Yaskawa INFORM job: SKRZYNIA_5240_180_STOPNI_10B_NEW.JBI

/JOB
//NAME SKRZYNIA_5240_180_STOPNI_10B_NEW
///FOLDERNAME 02-SKRZYNIE_JOBS
//POS
///NPOS 773,773,0,34,0,0
///TOOL 0
///POSTYPE PULSE
///PULSE
C00000=-21231,-51303,42314,2367,6591,-1439
C00001=-12854,-61498,-6635,149088,-29435,16513
C00002=84284,-61498,-6635,149088,14842,16513
C00003=84426,-61498,-62039,149088,14842,16513
C00004=84426,-61498,-83719,149088,14842,16513
C00005=40079,-25830,-61904,72398,37828,17494
C00006=40079,-25830,-61904,72398,37828,17494
C00007=38824,-23395,-60038,72349,38727,17731
C00008=41545,-22667,-59464,70826,37145,18191
C00009=40079,-25830,-61904,72398,37828,17494
C00010=40079,-23879,-31232,97616,36989,2612
C00011=40241,-22903,-30855,97033,36795,2952
C00012=39596,-21803,-29985,96678,37187,3182
C00013=41542,-21522,-29763,96797,35874,3054
C00014=40241,-22903,-30855,97033,36795,2952
C00015=44500,-22967,-34027,49689,40772,15208
C00016=44759,-21950,-33222,49364,40770,15399
C00017=43898,-20603,-32137,49608,41392,15289
C00018=45676,-20288,-31878,48567,40497,15854
C00019=44759,-21950,-33222,49364,40770,15399
C00020=50639,-31838,-53853,40430,42590,20636
C00021=47737,-42531,-47731,84740,46626,-3202
C00022=73324,-51450,-15857,136644,48513,-27329
C00023=28578,-31257,-33285,101874,54895,-3139
C00024=29101,-23166,-41439,93785,52323,3372
C00025=30342,-16402,-40775,90158,51109,6027
C00026=29555,-14242,-38855,90054,51607,6222
C00027=31304,-14182,-38798,89754,50458,6198
C00028=30342,-16402,-40775,90158,51109,6027
C00029=37840,-26567,-47806,97824,39338,5403
C00030=38314,-22656,-45541,96192,38787,6352
C00031=38740,-21749,-44817,95954,38481,6451
C00032=38106,-20505,-43805,95701,38856,6673
C00033=39920,-20274,-43616,95549,37666,6573
C00034=38740,-21749,-44817,95954,38481,6451
C00035=35154,-23288,-28184,89821,43405,2441
C00036=35403,-21021,-26397,89340,43215,2751
C00037=34678,-19569,-25213,89063,43699,2948
C00038=36545,-19419,-25091,89018,42427,2940
C00039=35403,-21021,-26397,89340,43215,2751
C00040=46673,-28267,-59493,36306,49500,22578
C00041=47298,-25083,-54483,36432,48421,22382
C00042=46134,-23276,-53085,36983,49197,22170
C00043=48093,-22778,-52692,35651,48513,22818
C00044=47298,-25083,-54483,36432,48421,22382
C00045=43000,-32780,-49011,53703,41088,15214
C00046=66148,-65994,-55487,105361,28212,-7739
C00047=66148,-65994,-55487,105361,28212,-7739
C00048=59848,-54778,-49507,133915,29212,-10807
C00049=45497,-38347,-41839,114412,32622,-465
C00050=46376,-32635,-46933,102993,29107,5780
C00051=46303,-28031,-46898,97061,28371,8976
C00052=45038,-26161,-45521,96183,29128,9541
C00053=46946,-25787,-45238,96120,27855,9431
C00054=46303,-28031,-46898,97061,28371,8976
C00055=45864,-17128,1685,129467,40696,-9274
C00056=46023,-15894,1830,128891,40053,-8896
C00057=45181,-14790,2774,128176,40341,-8535
C00058=46921,-14545,2986,129317,39465,-9073
C00059=45402,-17127,796,128656,40504,-8810
C00060=42828,-21985,-11573,106778,34538,-1929
C00061=43349,-21404,-11124,106831,34165,-1930
C00062=42250,-19876,-9917,105946,34757,-1485
C00063=44494,-19460,-9583,106781,33302,-1837
C00064=42797,-21858,-11474,106726,34550,-1903
C00065=42956,-14057,7354,88292,32197,-569
C00066=43438,-13569,7781,88275,31880,-510
C00067=42549,-12302,8904,87823,32462,-349
C00068=44721,-11883,9282,88161,31033,-316
C00069=42944,-14884,6642,88491,32210,-682
C00070=42956,-14057,7354,88292,32197,-569
C00071=43438,-13569,7781,88275,31880,-510
C00072=42549,-12302,8904,87823,32462,-349
C00073=44721,-11883,9282,88161,31033,-316
C00074=42944,-14884,6642,88491,32210,-682
C00075=42492,-36415,-29790,92406,42740,11684
C00076=29699,-14901,-14062,86637,51249,15251
C00077=28921,-12904,-12269,86425,51786,15406
C00078=30978,-12767,-12144,86426,50380,15429
C00079=29506,-17416,-16239,86937,51377,15018
C00080=29523,-100,37175,104016,54946,1530
C00081=29670,3692,41450,104134,54886,1470
C00082=29289,4768,42714,104010,55127,1477
C00083=31025,4720,42655,104739,54116,1295
C00084=29634,3577,41316,104108,54910,1473
C00085=88410,-69609,-60867,139529,19008,-8209
C00086=82254,-59190,-37505,135829,26015,-2584
C00087=48709,-26647,-10027,118963,31871,904
C00088=44740,-24992,-19428,105622,30913,8023
C00089=35836,-10089,175,120717,54219,3716
C00090=33571,-11609,-5533,116057,52820,8482
C00091=32638,-9483,-3533,115639,53262,8773
C00092=34483,-9329,-3384,116184,52162,8425
C00093=33571,-11609,-5533,116057,52820,8482
C00094=29299,-14235,-8112,85858,51306,13749
C00095=30258,-13056,-7056,85778,50658,13854
C00096=29454,-11053,-5212,85557,51212,13988
C00097=31306,-10982,-5149,85624,49953,14016
C00098=30258,-13056,-7056,85778,50658,13854
C00099=44150,-27478,-14760,79983,38437,11062
C00100=60260,-41997,-20174,82745,25327,6782
C00101=62412,-62489,-12046,-12266,17816,34850
C00102=0,-52280,40443,0,6876,0
C00103=-681,-52632,38645,-5695,5489,-631
C00104=-17840,-61498,-6635,-149088,-29435,-16513
C00105=-84284,-61498,-6635,-149088,14842,-16513
C00106=-84426,-61498,-62039,-149088,14842,-16513
C00107=-84426,-61498,-83719,-149088,14842,-16513
C00108=-83351,-27062,-60322,-167360,37385,6517
C00109=-83351,-27062,-60322,-167360,37385,23281
C00110=-45097,-23850,-79932,-76262,26943,-22849
C00111=-48253,-15729,-73342,-71138,25693,-24842
C00112=-50302,-13076,-73239,-65836,25323,-27140
C00113=-49401,-11675,-71961,-66260,25816,-27133
C00114=-50608,-11574,-71867,-65226,25249,-27391
C00115=-49660,-13361,-73494,-66442,25615,-26975
C00116=-48242,-21102,-77802,-73044,25430,-23851
C00117=-42432,-29691,-46140,-101591,34194,-3953
C00118=-40467,-32259,-45349,-89481,35752,-6083
C00119=-35590,-22323,-38089,-87474,43148,-7978
C00120=-34853,-20780,-36847,-87247,43643,-8181
C00121=-37029,-20471,-36594,-86926,42180,-8224
C00122=-35503,-23333,-38886,-87700,43207,-7835
C00123=-41659,-25848,-37197,-61468,39541,-12344
C00124=-42019,-23363,-32043,-63110,38591,-11327
C00125=-41283,-22167,-31102,-63128,39154,-11341
C00126=-43189,-21868,-30866,-62281,38009,-11788
C00127=-40846,-25460,-35158,-62968,39555,-11455
C00128=-39561,-32409,-42051,-71473,38885,-9254
C00129=-88477,-67032,-53890,-125185,13082,17955
C00130=-90715,-66667,-50935,-152816,24533,28486
C00131=-30735,-26920,-32844,-95116,50209,-1071
C00132=-37180,-24683,-31930,-114741,47007,2943
C00133=-36407,-19634,-34656,-109847,45004,-453
C00134=-38352,-16604,-33863,-108521,43129,-1176
C00135=-37479,-14809,-32279,-108169,43576,-1482
C00136=-39395,-14487,-31992,-108361,42368,-1194
C00137=-37253,-18321,-35339,-108644,43916,-1187
C00138=-30948,-19486,-27368,-89515,49970,-2899
C00139=-32453,-17458,-25663,-89179,48933,-3088
C00140=-31896,-16151,-24534,-89028,49305,-3221
C00141=-33527,-16125,-24510,-88960,48196,-3202
C00142=-31291,-18911,-26892,-89421,49733,-2955
C00143=-32789,-14788,-10714,-75998,48642,-1904
C00144=-33953,-13481,-9550,-75758,47902,-2112
C00145=-33380,-12226,-8408,-75670,48319,-2157
C00146=-35020,-12164,-8351,-75529,47228,-2306
C00147=-33300,-14767,-10697,-75957,48300,-1949
C00148=-33300,-14767,-10697,-75957,48300,-1949
C00149=-33901,-13199,-7224,-76945,47663,-1266
C00150=-33178,-11617,-5779,-76815,48184,-1329
C00151=-35129,-11426,-5603,-76688,46886,-1497
C00152=-32900,-14718,-9841,-76444,48459,-1584
C00153=-46324,-38325,-53351,-48650,39022,-16558
C00154=-84678,-53272,-42524,-56273,5220,-14251
C00155=-79949,-57830,-54545,-43165,18800,-25262
C00156=-85199,-63426,-59279,-35356,8253,-25340
C00157=-43240,-40066,-69296,-76804,34492,-13950
C00158=-32352,-24302,-62495,-76398,48702,-17646
C00159=-33867,-19497,-59989,-74208,48202,-18898
C00160=-33043,-17469,-58279,-74274,48770,-19034
C00161=-35172,-17180,-58031,-73305,47532,-19251
C00162=-33150,-20833,-61090,-74721,48572,-18687
C00163=-32525,-19963,-22291,-97454,48417,-2656
C00164=-34479,-17146,-19937,-97221,47013,-2812
C00165=-33716,-15515,-18525,-96928,47480,-3025
C00166=-35357,-15455,-18472,-97073,46375,-2908
C00167=-33341,-18474,-21063,-97306,47817,-2759
C00168=-32838,-10388,7981,-94473,48357,2926
C00169=-33747,-9461,8037,-94117,47673,2571
C00170=-33094,-8062,9377,-93861,48090,2458
C00171=-34952,-7927,9507,-94260,46861,2543
C00172=-33010,-10379,7174,-94037,48174,2591
C00173=-36099,-20774,-22249,-70758,44565,-7624
C00174=-37926,-16067,-12890,-73276,42575,-5996
C00175=-37323,-14944,-11908,-73188,43017,-6038
C00176=-39053,-14785,-11769,-72915,41882,-6255
C00177=-37847,-19214,-17221,-72670,42783,-6386
C00178=-36099,-20774,-22249,-70758,44565,-7624
C00179=-37926,-16067,-12890,-73276,42575,-5996
C00180=-37323,-14944,-11908,-73188,43017,-6038
C00181=-39053,-14785,-11769,-72915,41882,-6255
C00182=-37847,-19214,-17221,-72670,42783,-6386
C00183=-36099,-20774,-22249,-70758,44565,-7624
C00184=-37926,-16067,-12890,-73276,42575,-5996
C00185=-37323,-14944,-11908,-73188,43017,-6038
C00186=-39053,-14785,-11769,-72915,41882,-6255
C00187=-37847,-19214,-17221,-72670,42783,-6386
C00188=-37874,14907,75180,-111692,46453,18697
C00189=-37834,19259,81880,-112749,47050,19446
C00190=-37304,21381,85363,-113034,47644,19820
C00191=-39330,21904,86247,-114552,46854,20222
C00192=-38061,19744,82664,-113035,47027,19575
C00193=-73757,-59015,-49060,-81128,17325,-3444
C00194=-59391,-59726,-723,-139936,47315,26256
C00195=-59391,-63256,-7305,-138930,45803,25558
C00196=-41911,-25348,-18707,-96909,37821,5942
C00197=-39278,-18921,-13723,-94727,39374,4724
C00198=-50267,-3803,20766,-145166,53580,20077
C00199=-49199,-2294,22340,-144514,53890,19722
C00200=-50839,-1881,22778,-145489,53339,20243
C00201=-50267,-457,30009,-146420,56926,21139
C00202=-39278,-18921,-13723,-94727,39374,4724
C00203=-38355,-17353,-12416,-94258,39960,4466
C00204=-40180,-17161,-12255,-94505,38724,4557
C00205=-37963,-22229,-16363,-95272,40353,5112
C00206=-56568,-73357,-35482,-123268,35826,13545
C00207=-46099,-67236,-11725,-98004,28606,19827
C00208=275,-40498,62911,330,272,-175
C00209=-21231,-51303,42314,2367,6591,-1439
C00210=-12854,-61498,-6635,149088,-29435,16513
C00211=84284,-61498,-6635,149088,14842,16513
C00212=84426,-61498,-62039,149088,14842,16513
C00213=84426,-61498,-83719,149088,14842,16513
C00214=40079,-25830,-61904,72398,37828,17494
C00215=38665,-12403,-32409,107781,42694,-4781
C00216=38665,-12616,-38699,103566,41336,-2086
C00217=40079,-23879,-31232,97616,36989,2612
C00218=41034,-22333,-61710,53029,45515,35529
C00219=41034,-23109,-56119,56672,43067,33108
C00220=40241,-22903,-30855,97033,36795,2952
C00221=44500,-24561,-52671,41420,48760,20730
C00222=37674,-15115,-44130,49660,57471,17042
C00223=37674,-15093,-37691,51888,54769,15111
C00224=44759,-23105,-42292,45130,44325,18129
C00225=50639,-31838,-53853,40430,42590,20636
C00226=47737,-42531,-47731,84740,46626,-3202
C00227=78713,-49095,-28754,133607,38203,-24422
C00228=28578,-31257,-33285,101874,54895,-3139
C00229=29101,-23166,-41439,93785,52323,3372
C00230=31163,-13587,-30677,93779,50972,3168
C00231=31163,-14026,-37120,90592,50610,5586
C00232=30342,-16304,-38140,91492,51220,5006
C00233=37840,-26567,-47806,97824,39338,5403
C00234=38314,-22656,-45541,96192,38787,6352
C00235=39658,-19732,-37407,100215,38572,3786
C00236=39658,-20175,-43840,95284,37805,6758
C00237=38740,-21749,-44817,95954,38481,6451
C00238=35154,-25126,-38164,84243,43431,6092
C00239=35628,-20373,-48281,63877,49123,23186
C00240=35628,-20245,-42140,67132,47541,20849
C00241=35403,-21021,-26397,89340,43215,2751
C00242=46673,-26636,-70072,32738,56435,25418
C00243=35383,-13840,-53792,49898,63478,22502
C00244=35383,-14670,-48593,51546,60904,20775
C00245=47298,-24788,-58951,34834,51068,23565
C00246=43000,-32780,-49011,53703,41088,15214
C00247=90538,-65158,-52413,145953,6697,-22013
C00248=90538,-65158,-52413,145953,6697,-22013
C00249=59848,-54778,-49507,133915,29212,-10807
C00250=45497,-38347,-41839,114412,32622,-465
C00251=46376,-32635,-46933,102993,29107,5780
C00252=33967,-11360,-33206,103445,48358,510
C00253=33967,-11425,-39323,99951,47288,2995
C00254=46303,-28031,-46898,97061,28371,8976
C00255=45864,-24383,-22135,118487,33937,-2761
C00256=34441,-6148,1727,116719,55152,-8810
C00257=34441,-8494,-7364,114007,52974,-6586
C00258=45402,-26628,-33163,110407,31435,1774
C00259=42828,-30834,-56687,70923,33806,18230
C00260=32432,-16862,-57229,61149,56469,35022
C00261=32432,-17753,-51657,63804,54519,32761
C00262=42797,-29457,-43215,82997,32293,11437
C00263=42956,-27250,-43688,55004,39651,18538
C00264=34828,-16613,-38353,58296,54652,20387
C00265=34828,-16027,-31548,60910,52619,18267
C00266=33058,-19049,-34141,61806,53461,17709
C00267=33058,-12296,-3124,73891,47808,8644
C00268=33058,-12296,-3124,73891,47808,8644
C00269=34828,-9500,-717,73395,46757,9098
C00270=34828,-6540,9127,77476,45790,6283
C00271=33897,-9329,6906,77965,46306,5856
C00272=33897,-9329,6906,77965,46306,5856
C00273=34828,-9385,-322,73557,46711,8985
C00274=34828,-6437,9450,77608,45767,6193
C00275=34037,-8372,7553,77721,46264,6039
C00276=34037,3206,39942,90427,45468,-2620
C00277=34037,-4564,18961,82315,45612,2890
C00278=34657,-86,29234,85939,44999,527
C00279=34657,5122,42910,91205,45125,-3022
C00280=29506,-17416,-16239,86937,51377,15018
C00281=88410,-69609,-60867,139529,19008,-8209
C00282=82254,-59190,-37505,135829,26015,-2584
C00283=48709,-26647,-10027,118963,31871,904
C00284=44740,-24992,-19428,105622,30913,8023
C00285=35836,-628,28594,126575,61828,-1622
C00286=32584,7682,39174,123909,66904,-2731
C00287=32584,2860,25722,121968,63529,-448
C00288=33571,-6628,11088,120434,56899,4821
C00289=29299,-14235,-8112,85858,51306,13749
C00290=31207,-8871,1432,87980,49993,12258
C00291=31207,-5884,11163,91534,50189,9605
C00292=30258,-13056,-7056,85778,50658,13854
C00293=44150,-27478,-14760,79983,38437,11062
C00294=60260,-41997,-20174,82745,25327,6782
C00295=62412,-62489,-12046,-12266,17816,34850
C00296=0,-52280,40443,0,6876,0
C00297=-681,-52632,38645,-5695,5489,-631
C00298=-17840,-61498,-6635,-149088,-29435,-16513
C00299=-84284,-61498,-6635,-149088,14842,-16513
C00300=-84426,-61498,-62039,-149088,14842,-16513
C00301=-84426,-61498,-83719,-149088,14842,-16513
C00302=-83351,-27062,-60322,-167360,37385,6517
C00303=-83351,-27062,-60322,-167360,37385,23281
C00304=-45097,-23850,-79932,-76262,26943,-22849
C00305=-48253,-15729,-73342,-71138,25693,-24842
C00306=-42968,-5377,-68871,-73541,34127,-27123
C00307=-42968,-1764,-72258,-66870,35661,-30967
C00308=-49660,-13361,-73494,-66442,25615,-26975
C00309=-48242,-21102,-77802,-73044,25430,-23851
C00310=-42432,-29691,-46140,-101591,34194,-3953
C00311=-40467,-32259,-45349,-89481,35752,-6083
C00312=-32572,-16306,-55553,-67397,53381,-30018
C00313=-32572,-17083,-50158,-70353,51979,-27676
C00314=-35503,-23333,-38886,-87700,43207,-7835
C00315=-41659,-27404,-51576,-53376,44034,-17488
C00316=-31493,-12293,-40596,-60462,61580,-18646
C00317=-31493,-12246,-34421,-62460,59687,-16660
C00318=-40846,-26766,-43924,-57962,41907,-14588
C00319=-39561,-32409,-42051,-71473,38885,-9254
C00320=-88477,-67032,-53890,-125185,13082,17955
C00321=-90715,-66667,-50935,-152816,24533,28486
C00322=-30735,-26920,-32844,-95116,50209,-1071
C00323=-37180,-24683,-31930,-114741,47007,2943
C00324=-36407,-19634,-34656,-109847,45004,-453
C00325=-39265,-13210,-22525,-113458,44747,2144
C00326=-39265,-14219,-29616,-109727,42998,-318
C00327=-37253,-17754,-30753,-111100,44998,450
C00328=-30948,-19486,-27368,-89515,49970,-2899
C00329=-32883,-16993,-41795,-70354,52410,-19465
C00330=-32883,-16648,-35340,-73373,51262,-17121
C00331=-31291,-18911,-26892,-89421,49733,-2955
C00332=-32789,-18082,-25081,-70149,50526,-6217
C00333=-30947,-8963,-19167,-66964,58291,-13111
C00334=-30947,-7534,-11276,-69435,56821,-10881
C00335=-33300,-16430,-17409,-73196,49065,-3948
C00336=-33300,-18454,-27193,-69159,50560,-6941
C00337=-29440,-7196,-21034,-66741,61979,-14499
C00338=-29440,-6022,-13253,-68913,60441,-12298
C00339=-32900,-16744,-17947,-73145,49365,-3984
C00340=-46324,-38325,-53351,-48650,39022,-16558
C00341=-84678,-53272,-42524,-56273,5220,-14251
C00342=-79949,-57830,-54545,-43165,18800,-25262
C00343=-85199,-63426,-59279,-35356,8253,-25340
C00344=-43240,-40066,-69296,-76804,34492,-13950
C00345=-32352,-24302,-62495,-76398,48702,-17646
C00346=-32091,-8283,-47690,-89191,50586,-9020
C00347=-32091,-6854,-52880,-85538,50580,-11777
C00348=-33150,-19215,-66726,-70659,49900,-21662
C00349=-32525,-23315,-42550,-87560,47339,-9680
C00350=-33177,-11430,-23623,-100299,50817,3381
C00351=-33177,-12228,-30638,-97022,49957,920
C00352=-33341,-22016,-46198,-84312,46879,-11867
C00353=-32838,-21830,-40242,-73680,49831,-12021
C00354=-32060,-14432,-37779,-68594,55292,-20152
C00355=-32060,-13998,-31234,-71279,54006,-17916
C00356=-32826,-17642,-34445,-71437,53361,-17708
C00357=-36099,-24001,-62103,-52600,56003,-20988
C00358=-33061,-10268,-52363,-54704,65882,-25434
C00359=-33061,-11342,-46906,-56402,63410,-23481
C00360=-32436,-13964,-49327,-56793,63580,-23241
C00361=-36099,-22018,-27900,-68071,45501,-9434
C00362=-33133,-10810,-21932,-64736,55524,-15558
C00363=-33133,-9463,-14247,-67406,53929,-13330
C00364=-32817,-11797,-16457,-67620,54048,-13161
C00365=-36099,-9367,15363,-88420,42122,3838
C00366=-33275,421,22196,-80432,49557,-3328
C00367=-33275,4923,34904,-84824,49106,-106
C00368=-32887,2565,32173,-84656,49359,-162
C00369=-32887,2565,32173,-84656,49359,-162
C00370=-33016,5847,38022,-85966,49224,775
C00371=-33016,12470,54924,-91440,49393,4788
C00372=-31218,6775,44553,-88539,50343,3051
C00373=-82794,-53123,-36553,-147152,20085,23769
C00374=-59391,-59726,-723,-139936,47315,26256
C00375=-59391,-69594,-18878,-137021,43274,24283
C00376=-41911,-25348,-18707,-96909,37821,5942
C00377=-39278,-18921,-13723,-94727,39374,4724
C00378=-42007,14667,57624,-137771,70069,18031
C00379=-42007,7816,40199,-136118,64730,15895
C00380=-50267,-457,30009,-146420,56926,21139
C00381=-32199,-12839,-21112,-74266,52126,-18055
C00382=-32186,-11312,-13395,-77340,51278,-15674
C00383=-37963,-22229,-16363,-95272,40353,5112
C00384=-66368,-73811,-34662,-141094,38161,28545
C00385=-46099,-67236,-11725,-98004,28606,19827
C00386=275,-40498,62911,330,272,-175
C00387=-21231,-51303,42314,2367,6591,-1439
C00388=-12854,-61498,-6635,149088,-29435,16513
C00389=32880,-72586,-50560,79734,53940,25582
C00390=76664,-93599,-96338,114349,24908,7990
C00391=72545,-76403,-90681,98079,12187,16258
C00392=68435,-42241,-79282,43384,21203,43145
C00393=65057,-16377,-54230,51764,24572,24912
C00394=65057,-16377,-54230,51764,24572,24912
C00395=63338,-14509,-52578,53100,25585,24479
C00396=65493,-13068,-51269,50530,24633,25485
C00397=65057,-16377,-54230,51764,24572,24912
C00398=65057,-15356,-24189,99795,20011,765
C00399=64877,-14372,-23690,98704,20045,1316
C00400=64002,-13489,-22890,98156,20604,1621
C00401=65592,-12702,-22173,98357,19527,1466
C00402=64877,-14372,-23690,98704,20045,1316
C00403=68341,-13254,-25781,29903,31229,25524
C00404=68283,-12212,-24821,29865,31356,25548
C00405=67188,-11145,-23825,30867,31841,25051
C00406=68624,-10377,-23095,29361,31405,25809
C00407=68283,-12212,-24821,29865,31356,25548
C00408=67373,-28813,-51747,26561,36937,27500
C00409=65665,-56911,-59086,75825,31170,1181
C00410=86238,-56758,-47218,93606,16664,-7096
C00411=86238,-56758,-47218,93606,16664,-7096
C00412=58162,-25487,-29222,106212,35121,-6052
C00413=54729,-17550,-36821,90686,35172,3055
C00414=53879,-10723,-35593,84994,35691,6442
C00415=52628,-8898,-33837,85063,36512,6546
C00416=54193,-8333,-33282,84633,35489,6620
C00417=53879,-10723,-35593,84994,35691,6442
C00418=63265,-18185,-41125,95483,22448,4389
C00419=62561,-14368,-38517,92984,22773,5727
C00420=62689,-13396,-37636,92694,22678,5861
C00421=61812,-12400,-36718,92465,23238,6064
C00422=63331,-11679,-36046,92201,22238,6052
C00423=62689,-13396,-37636,92694,22678,5861
C00424=60836,-16142,-22303,87853,25853,3109
C00425=60346,-13901,-20318,87240,26185,3441
C00426=59279,-12702,-19226,86999,26911,3593
C00427=60868,-12050,-18626,86765,25831,3679
C00428=60346,-13901,-20318,87240,26185,3441
C00429=71174,-16943,-50501,16787,44328,31924
C00430=70846,-13961,-45205,17496,43056,31510
C00431=69412,-12602,-43961,18675,43507,30969
C00432=70949,-11616,-43043,17320,43301,31610
C00433=70846,-13961,-45205,17496,43056,31510
C00434=66765,-25643,-43957,33958,30926,25005
C00435=89904,-51519,-74342,14421,36812,44678
C00436=59533,-60921,-66479,83565,41795,11392
C00437=74572,-27669,-34920,136415,14797,-11887
C00438=72479,-21736,-38943,108586,11547,1590
C00439=70901,-17325,-38411,94105,11830,8638
C00440=69318,-15905,-37172,92885,12849,9347
C00441=70820,-15051,-36412,92531,11846,9399
C00442=70901,-17325,-38411,94105,11830,8638
C00443=70927,-7523,10343,151197,29871,-19432
C00444=70517,-6236,10737,150221,29352,-18933
C00445=69462,-5331,11645,148944,29606,-18324
C00446=70849,-4645,12343,150548,29173,-19084
C00447=70402,-7634,9356,150158,29478,-18907
C00448=68660,-13051,-4106,122816,18275,-8999
C00449=68895,-12351,-3471,122899,18094,-9031
C00450=67458,-11121,-2337,120787,18802,-8043
C00451=69212,-10147,-1425,122703,17774,-8922
C00452=68590,-12934,-4000,122687,18305,-8939
C00453=67960,-5141,15741,92957,15720,-628
C00454=68207,-4523,16370,92944,15555,-601
C00455=67051,-3465,17460,92338,16311,-404
C00456=68762,-2475,18496,92897,15183,-531
C00457=68227,-5981,14898,93242,15553,-745
C00458=67960,-5141,15741,92957,15720,-628
C00459=68207,-4523,16370,92944,15555,-601
C00460=67051,-3465,17460,92338,16311,-404
C00461=68762,-2475,18496,92897,15183,-531
C00462=68227,-5981,14898,93242,15553,-745
C00463=67960,-5141,15741,92957,15720,-628
C00464=68207,-4523,16370,92944,15555,-601
C00465=67051,-3465,17460,92338,16311,-404
C00466=68762,-2475,18496,92897,15183,-531
C00467=68227,-5981,14898,93242,15553,-745
C00468=67960,-5141,15741,92957,15720,-628
C00469=68207,-4523,16370,92944,15555,-601
C00470=67051,-3465,17460,92338,16311,-404
C00471=68762,-2475,18496,92897,15183,-531
C00472=68227,-5981,14898,93242,15553,-745
C00473=89016,-59505,-36896,143842,20811,-11822
C00474=60495,-76741,-47652,120298,37447,-3273
C00475=76037,-16315,-2108,148598,17507,-12246
C00476=70560,-15452,-11753,122116,14270,428
C00477=59169,-3122,7113,131317,41741,-2292
C00478=57131,-5277,619,125436,39242,3005
C00479=55729,-3443,2508,124592,39934,3479
C00480=57337,-2775,3210,125461,39069,2998
C00481=57131,-5277,619,125436,39242,3005
C00482=54062,-9026,-3291,86300,34474,14396
C00483=54568,-7612,-1915,86151,34132,14497
C00484=53276,-5879,-187,85948,35014,14576
C00485=54919,-5291,406,85945,33897,14626
C00486=54568,-7612,-1915,86151,34132,14497
C00487=55516,-30048,-16468,81245,30784,11190
C00488=78642,-41617,-20006,83725,13431,8209
C00489=0,-52280,40443,0,6876,0
C00490=-681,-52632,38645,-5695,5489,-631
C00491=-17840,-61498,-6635,-149088,-29435,-16513
C00492=-84284,-61498,-6635,-149088,14842,-16513
C00493=-57949,-92832,-68327,-119114,39180,-13331
C00494=-51160,-78996,-68705,-103851,38676,-21739
C00495=-70129,-12201,-70194,-45988,15849,-32683
C00496=-70861,-4247,-62448,-43170,16032,-33903
C00497=-72229,-1292,-61598,-37253,16795,-36501
C00498=-71164,-286,-60510,-39045,17142,-35862
C00499=-72168,114,-60071,-37345,16819,-36474
C00500=-71747,-1710,-62044,-38091,16943,-36199
C00501=-72086,-8949,-67137,-41785,15362,-34318
C00502=-68226,-19972,-38714,-103620,16923,-1218
C00503=-67549,-22986,-38612,-80975,17520,-9124
C00504=-60286,-14955,-31870,-81576,26630,-9634
C00505=-59206,-13694,-30736,-81541,27366,-9725
C00506=-61026,-12796,-29913,-80837,26167,-9971
C00507=-60502,-15936,-32740,-81790,26471,-9505
C00508=-66711,-16726,-29834,-42060,26790,-21996
C00509=-66477,-14329,-24475,-44917,25565,-20507
C00510=-65503,-13376,-23611,-45716,26132,-20127
C00511=-67048,-12587,-22889,-44009,25442,-20959
C00512=-66009,-16611,-27996,-44380,26285,-20808
C00513=-67084,-23473,-35621,-52822,22843,-18344
C00514=-54372,-63877,-56403,-90862,27079,1323
C00515=-55608,-75012,-34654,-126966,55573,20814
C00516=-55608,-75012,-34654,-126966,55573,20814
C00517=-58069,-20780,-28125,-95622,31565,-134
C00518=-62818,-16895,-25617,-123146,31403,8811
C00519=-60301,-12189,-28106,-114654,29999,4030
C00520=-61167,-8731,-26593,-112607,28768,2985
C00521=-59960,-7252,-25135,-111997,29446,2563
C00522=-61574,-6413,-24296,-112502,28453,2957
C00523=-60636,-10677,-28466,-112685,29164,2987
C00524=-55814,-13636,-22293,-87541,33030,-3263
C00525=-56566,-11270,-20110,-87077,32519,-3496
C00526=-55709,-10167,-19066,-86969,33101,-3589
C00527=-57154,-9687,-18605,-86794,32120,-3632
C00528=-55949,-12989,-21706,-87412,32939,-3330
C00529=-57109,-8613,-4995,-71756,32687,-5152
C00530=-57764,-7017,-3429,-71410,32292,-5358
C00531=-56909,-5946,-2356,-71529,32873,-5273
C00532=-58347,-5433,-1836,-71115,31941,-5534
C00533=-57555,-8453,-4841,-71622,32398,-5235
C00534=-57555,-8453,-4841,-71622,32398,-5235
C00535=-57844,-6749,-1100,-73475,31868,-4209
C00536=-56760,-5394,262,-73573,32605,-4123
C00537=-58439,-4668,1002,-73167,31507,-4396
C00538=-57269,-8513,-4090,-72514,32435,-4729
C00539=-74194,-26905,-45748,-21164,30431,-30370
C00540=-93036,-61583,-83098,-4972,39040,-38907
C00541=-93036,-61583,-83098,-4972,39040,-38907
C00542=-71878,-28414,-61729,-48672,19032,-25171
C00543=-58025,-17185,-56692,-61796,34178,-22014
C00544=-58138,-12270,-53641,-59720,34855,-23185
C00545=-56898,-10637,-52111,-60384,35596,-23031
C00546=-58712,-9745,-51261,-58987,34681,-23500
C00547=-57851,-13714,-54968,-60141,34926,-22995
C00548=-57767,-13689,-16896,-100181,31334,-836
C00549=-58645,-10437,-13885,-99794,30663,-1040
C00550=-57513,-9065,-12573,-99347,31388,-1300
C00551=-58947,-8556,-12078,-99591,30423,-1148
C00552=-58031,-12031,-15383,-99926,31110,-974
C00553=-57646,-4162,14084,-101426,32077,4804
C00554=-58050,-2999,14481,-100683,31666,4357
C00555=-57067,-1784,15765,-100255,32298,4198
C00556=-58672,-1130,16464,-100866,31256,4407
C00557=-57676,-4116,13320,-100600,31921,4338
C00558=-61201,-13510,-16039,-60848,29053,-13371
C00559=-61885,-8475,-5914,-65722,27292,-10768
C00560=-61040,-7537,-4993,-65975,27855,-10622
C00561=-62506,-6917,-4380,-65230,26947,-11038
C00562=-62587,-11561,-10517,-63923,27184,-11731
C00563=-61201,-13510,-16039,-60848,29053,-13371
C00564=-61885,-8475,-5914,-65722,27292,-10768
C00565=-61040,-7537,-4993,-65975,27855,-10622
C00566=-62506,-6917,-4380,-65230,26947,-11038
C00567=-62587,-11561,-10517,-63923,27184,-11731
C00568=-61201,-13510,-16039,-60848,29053,-13371
C00569=-61885,-8475,-5914,-65722,27292,-10768
C00570=-61040,-7537,-4993,-65975,27855,-10622
C00571=-62506,-6917,-4380,-65230,26947,-11038
C00572=-62587,-11561,-10517,-63923,27184,-11731
C00573=-61201,-13510,-16039,-60848,29053,-13371
C00574=-61885,-8475,-5914,-65722,27292,-10768
C00575=-61040,-7537,-4993,-65975,27855,-10622
C00576=-62506,-6917,-4380,-65230,26947,-11038
C00577=-62587,-11561,-10517,-63923,27184,-11731
C00578=-66017,-67071,-29713,-134523,32873,22112
C00579=-66017,-67071,-29713,-134523,48860,22112
C00580=-66017,-67071,-29713,-134523,48860,22112
C00581=-68464,-16512,-11702,-102583,19802,8050
C00582=-64069,-10918,-6685,-98748,22529,6223
C00583=-71808,7543,33524,-159735,48317,27747
C00584=-70546,8877,35161,-158835,48660,27285
C00585=-71854,9797,36309,-159820,48523,27800
C00586=-71808,11433,44144,-160620,52560,28413
C00587=-64069,-10918,-6685,-98748,22529,6223
C00588=-62794,-9626,-5461,-98007,23355,5872
C00589=-64311,-8958,-4821,-98397,22329,6039
C00590=-64031,-14482,-9933,-99750,22651,6736
C00591=-78219,-66180,-35295,-149347,29259,30999
C00592=-46099,-67236,-11725,-98004,28606,19827
C00593=275,-40498,62911,330,272,-175
C00594=-21231,-51303,42314,2367,6591,-1439
C00595=-12854,-61498,-6635,149088,-29435,16513
C00596=84284,-61498,-6635,149088,14842,16513
C00597=84426,-61498,-62039,149088,14842,16513
C00598=84426,-61498,-83719,149088,14842,16513
C00599=65057,-16377,-54230,51764,24572,24912
C00600=84041,-13116,-46066,-44825,8720,68452
C00601=84041,-13116,-46066,-44825,8720,68452
C00602=65057,-15356,-24189,99795,20011,765
C00603=67637,-3172,7568,143600,31056,-30644
C00604=67662,-5608,-1431,139396,27428,-28372
C00605=64877,-14372,-23690,98704,20045,1316
C00606=68341,-14112,-46560,22080,43478,30152
C00607=74439,-12048,-42441,10496,39800,35438
C00608=74439,-12165,-36552,11511,35735,34830
C00609=68283,-13111,-33582,26121,36053,27673
C00610=75452,-19560,-44582,17787,36745,31835
C00611=68183,-44834,-62310,40554,34116,19994
C00612=94103,-63119,-69903,16230,17694,31762
C00613=91219,-55958,-51219,93435,14423,-1742
C00614=58162,-25487,-29222,106212,35121,-6052
C00615=54729,-17550,-36821,90686,35172,3055
C00616=66899,-10128,-18429,123667,21445,-19920
C00617=66899,-11189,-25619,114518,19187,-15337
C00618=53879,-10723,-35593,84994,35691,6442
C00619=63265,-18185,-41125,95483,22448,4389
C00620=62561,-13957,-31618,102858,23622,675
C00621=69590,-4213,-7839,146392,28217,-29211
C00622=69590,-5671,-16037,141735,24331,-26767
C00623=62689,-13396,-37636,92694,22678,5861
C00624=60836,-16142,-22303,87853,25853,3109
C00625=70419,-6792,3293,145112,24366,-34895
C00626=70419,-9347,-6132,139211,20547,-31894
C00627=60346,-13901,-20318,87240,26185,3441
C00628=71174,-14707,-61072,14672,52947,33449
C00629=74702,-3968,-57019,7246,61374,46383
C00630=74702,-6026,-52329,7608,56632,46043
C00631=70846,-13961,-45205,17496,43056,31510
C00632=69645,-22678,-41665,30358,30421,26767
C00633=81017,-78801,-66317,80675,7786,2447
C00634=81017,-78801,-66317,80675,7786,2447
C00635=74572,-27669,-34920,136415,14797,-11887
C00636=72479,-22242,-45651,87952,10699,11452
C00637=69672,-10832,-32642,120831,15984,-9730
C00638=69672,-10902,-38542,108009,14088,-3499
C00639=70901,-17325,-38411,94105,11830,8638
C00640=70927,-14654,-14578,138497,19645,-12882
C00641=69868,-2819,8566,151833,34290,-26436
C00642=69868,-5527,-1288,148739,29985,-24711
C00643=70402,-15633,-20098,131974,17549,-9644
C00644=68660,-19736,-34792,69483,15374,16984
C00645=66723,-4601,3983,141012,31335,-31205
C00646=66723,-6984,-5147,136395,27741,-28704
C00647=68590,-19875,-36965,65038,15913,19153
C00648=67960,-17785,-38905,31205,30461,30184
C00649=81886,-7317,-45445,-3456,52807,41803
C00650=81886,-8115,-39300,-3703,47981,41989
C00651=68227,-16956,-25811,40505,23614,25262
C00652=67960,-17785,-38905,31205,30461,30184
C00653=81886,-7317,-45445,-3456,52807,41803
C00654=81886,-8115,-39300,-3703,47981,41989
C00655=68227,-16956,-25811,40505,23614,25262
C00656=67960,-17785,-38905,31205,30461,30184
C00657=81826,-7419,-45546,-3412,52798,41785
C00658=81848,-8180,-39364,-3674,47975,41975
C00659=68227,-16956,-25811,40505,23614,25262
C00660=67960,-17785,-38905,31205,30461,30184
C00661=81826,-7419,-45546,-3412,52798,41785
C00662=81841,-8193,-39376,-3669,47974,41973
C00663=71602,-15245,-36817,18211,35590,43873
C00664=46050,-47732,-32699,100114,41423,7030
C00665=72866,-68602,-36981,132032,32409,-7906
C00666=72866,-68602,-36981,132032,32409,-7906
C00667=76037,-16315,-2108,148598,17507,-12246
C00668=70560,-15452,-11753,122116,14270,428
C00669=59169,6935,37394,139131,51878,-7708
C00670=74026,19667,66991,167459,60328,-21429
C00671=74004,11336,46435,166776,52513,-20840
C00672=70596,-6436,10894,154825,32661,-13042
C00673=54062,-9026,-3291,86300,34474,14396
C00674=68545,-10695,-9472,57395,16045,33162
C00675=68545,-8345,-444,72070,14274,26026
C00676=54568,-3381,12592,95759,34582,9001
C00677=62643,-28068,-15160,80125,26114,12294
C00678=92151,-29067,-13111,41177,6909,29587
C00679=79691,-50270,-13176,-792,17881,39424
C00680=0,-52280,40443,0,6876,0
C00681=-681,-52632,38645,-5695,5489,-631
C00682=-17840,-61498,-6635,-149088,-29435,-16513
C00683=-84284,-61498,-6635,-149088,14842,-16513
C00684=-84426,-61498,-62039,-149088,14842,-16513
C00685=-84426,-61498,-83719,-149088,14842,-16513
C00686=-83351,-27062,-60322,-167360,37385,6517
C00687=-83351,-27062,-60322,-167360,37385,23281
C00688=-70129,-12201,-70194,-45988,15849,-32683
C00689=-70861,-4247,-62448,-43170,16032,-33903
C00690=-76882,1581,-62692,-12385,17047,-46133
C00691=-76882,5115,-65815,-9764,21769,-47439
C00692=-71747,1973,-65943,-29402,21445,-40519
C00693=-72086,-8949,-67137,-41785,15362,-34318
C00694=-68226,-19972,-38714,-103620,16923,-1218
C00695=-67549,-22986,-38612,-80975,17520,-9124
C00696=-67571,-8767,-63845,-20857,47895,-51617
C00697=-67571,-11045,-59117,-22639,43294,-50403
C00698=-60502,-15936,-32740,-81790,26471,-9505
C00699=-66711,-17800,-45499,-31995,34681,-27503
C00700=-69746,-8324,-48192,-17464,49433,-41898
C00701=-69746,-9218,-42644,-18734,45170,-41005
C00702=-66009,-17835,-39148,-36467,31351,-25061
C00703=-61601,-28306,-39228,-59626,25389,-15050
C00704=-72315,-63222,-70224,-69600,33305,-10426
C00705=-72315,-63222,-70224,-69600,33305,-10426
C00706=-58069,-20780,-28125,-95622,31565,-134
C00707=-62818,-16895,-25617,-123146,31403,8811
C00708=-60301,-10327,-15966,-123744,33797,9078
C00709=-71086,-3839,-6738,-149148,28394,26564
C00710=-71086,-5266,-14457,-145255,24651,24516
C00711=-60636,-10125,-23433,-117195,30623,5441
C00712=-55814,-13636,-22293,-87541,33030,-3263
C00713=-69422,-12084,-52013,-20684,41500,-45223
C00714=-69422,-12981,-46262,-22760,37210,-43951
C00715=-54522,-12876,-36643,-58338,40688,-32753
C00716=-57109,-11909,-20196,-61151,35632,-11198
C00717=-66848,-9895,-26530,-31737,34609,-32232
C00718=-66848,-8979,-19361,-35344,31107,-30205
C00719=-57555,-8453,-4841,-71622,32398,-5235
C00720=-53440,-7746,-26914,-52653,48023,-23958
C00721=-66139,-8692,-33669,-27706,42592,-36915
C00722=-66139,-8415,-27171,-30073,38884,-35433
C00723=-57269,-12429,-22388,-59751,36057,-12009
C00724=-74194,-26905,-45748,-21164,30431,-30370
C00725=-76007,-77202,-67157,-59280,11041,-11579
C00726=-76006,-77203,-67157,-59281,11043,-11581
C00727=-53398,-42726,-55849,-45492,34374,-18069
C00728=-71878,-28414,-61729,-48672,19032,-25171
C00729=-58025,-15345,-63150,-54975,37089,-25981
C00730=-69888,-7800,-37440,-106422,14795,8904
C00731=-69888,-7229,-43099,-90296,13928,1094
C00732=-57851,-11642,-61296,-53542,38019,-26875
C00733=-57767,-16815,-39222,-79084,30774,-12406
C00734=-68009,-6777,-10785,-133676,25020,23861
C00735=-68009,-8214,-18879,-126468,21885,20166
C00736=-58031,-15036,-36781,-79552,30550,-12125
C00737=-57667,-14715,-27905,-75704,31620,-11137
C00738=-65584,-8415,-48570,-25889,47500,-45851
C00739=-65584,-9360,-42775,-27961,43332,-44446
C00740=-57676,-13472,-23570,-71775,32303,-11588
C00741=-61201,-15867,-54988,-36061,45747,-27848
C00742=-67076,-3052,-56612,-19718,60798,-44143
C00743=-67076,-5062,-52229,-20645,56559,-43278
C00744=-62587,-15962,-44655,-39719,39603,-25252
C00745=-61201,-15867,-54988,-36061,45747,-27848
C00746=-67076,-3052,-56612,-19718,60798,-44143
C00747=-67076,-5062,-52229,-20645,56559,-43278
C00748=-62587,-15962,-44655,-39719,39603,-25252
C00749=-61201,-15867,-54988,-36061,45747,-27848
C00750=-67076,-3052,-56612,-19718,60798,-44143
C00751=-67076,-5062,-52229,-20645,56559,-43278
C00752=-62587,-15962,-44655,-39719,39603,-25252
C00753=-61201,-15867,-54988,-36061,45747,-27848
C00754=-67076,-3052,-56612,-19718,60798,-44143
C00755=-67076,-5062,-52229,-20645,56559,-43278
C00756=-62587,-15962,-44655,-39719,39603,-25252
C00757=-65551,-48104,-28924,-114827,24376,11665
C00758=-39771,-60653,-24362,-111239,58263,14171
C00759=-39771,-60652,-24363,-111239,58260,14167
C00760=-68464,-16512,-11702,-102583,19802,8050
C00761=-64069,-10918,-6685,-98748,22529,6223
C00762=-65559,2888,28457,-143691,38768,45726
C00763=-71346,27670,74204,-161919,66685,34494
C00764=-71346,18414,51305,-160904,58125,33425
C00765=-71808,11433,44144,-160620,52560,28413
C00766=-74529,-11525,-8997,-111700,8518,12107
C00767=-69976,-13061,-30302,-28674,27690,-38623
C00768=-69976,-12185,-23289,-33056,24143,-36329
C00769=-64031,-14482,-9933,-99750,22651,6736
C00770=-65667,-47452,-26760,-125785,27682,20101
C00771=-46099,-67236,-11725,-98004,28606,19827
C00772=275,-40498,62911,330,272,-175
BC00000=467225
BC00001=513669
BC00002=494109
BC00003=467540
BC00004=467540
BC00005=478876
BC00006=478876
BC00007=478876
BC00008=478876
BC00009=478876
BC00010=471196
BC00011=471196
BC00012=471196
BC00013=471196
BC00014=471196
BC00015=460443
BC00016=460443
BC00017=460443
BC00018=460443
BC00019=460443
BC00020=478876
BC00021=481980
BC00022=563952
BC00023=606256
BC00024=606256
BC00025=612396
BC00026=612396
BC00027=612396
BC00028=612396
BC00029=654662
BC00030=654618
BC00031=657690
BC00032=657690
BC00033=657690
BC00034=657690
BC00035=648474
BC00036=648474
BC00037=648474
BC00038=648474
BC00039=648474
BC00040=674113
BC00041=674113
BC00042=674061
BC00043=674061
BC00044=674113
BC00045=652574
BC00046=648164
BC00047=761837
BC00048=784046
BC00049=784046
BC00050=784046
BC00051=765613
BC00052=765613
BC00053=765613
BC00054=765613
BC00055=756396
BC00056=756396
BC00057=756396
BC00058=756396
BC00059=756396
BC00060=784268
BC00061=784268
BC00062=784268
BC00063=784268
BC00064=784268
BC00065=778123
BC00066=778123
BC00067=778123
BC00068=778123
BC00069=778123
BC00070=816525
BC00071=816525
BC00072=816525
BC00073=816525
BC00074=816525
BC00075=895775
BC00076=895775
BC00077=895775
BC00078=895775
BC00079=895775
BC00080=875385
BC00081=890707
BC00082=890707
BC00083=890707
BC00084=890707
BC00085=915591
BC00086=1005127
BC00087=999652
BC00088=999652
BC00089=1007990
BC00090=1007827
BC00091=1007827
BC00092=1007827
BC00093=1007827
BC00094=998610
BC00095=998610
BC00096=998610
BC00097=998610
BC00098=998610
BC00099=981572
BC00100=972138
BC00101=892453
BC00102=828403
BC00103=518986
BC00104=509920
BC00105=467540
BC00106=467540
BC00107=467540
BC00108=521167
BC00109=520352
BC00110=535759
BC00111=535759
BC00112=535757
BC00113=535757
BC00114=535757
BC00115=535757
BC00116=535757
BC00117=485653
BC00118=476436
BC00119=476436
BC00120=476436
BC00121=476436
BC00122=476436
BC00123=471828
BC00124=471828
BC00125=471828
BC00126=471828
BC00127=471828
BC00128=485653
BC00129=485653
BC00130=615112
BC00131=615112
BC00132=624329
BC00133=624329
BC00134=624329
BC00135=624329
BC00136=624329
BC00137=624329
BC00138=615112
BC00139=615112
BC00140=615112
BC00141=615112
BC00142=615112
BC00143=615112
BC00144=608968
BC00145=608968
BC00146=608968
BC00147=608968
BC00148=645787
BC00149=645787
BC00150=645787
BC00151=645787
BC00152=645787
BC00153=655680
BC00154=643721
BC00155=643721
BC00156=793396
BC00157=782173
BC00158=782173
BC00159=782173
BC00160=782173
BC00161=782173
BC00162=782173
BC00163=768348
BC00164=768348
BC00165=768348
BC00166=768348
BC00167=768348
BC00168=760668
BC00169=760668
BC00170=760668
BC00171=760668
BC00172=760668
BC00173=799584
BC00174=799584
BC00175=799584
BC00176=799584
BC00177=799584
BC00178=837986
BC00179=837986
BC00180=837986
BC00181=837986
BC00182=837986
BC00183=876389
BC00184=876389
BC00185=876389
BC00186=876389
BC00187=876389
BC00188=852671
BC00189=861919
BC00190=861919
BC00191=861922
BC00192=861922
BC00193=845667
BC00194=862979
BC00195=977267
BC00196=1008066
BC00197=1008066
BC00198=1002748
BC00199=1002748
BC00200=1002748
BC00201=1002748
BC00202=1015746
BC00203=1015746
BC00204=1015746
BC00205=1015746
BC00206=991691
BC00207=895479
BC00208=639407
BC00209=467225
BC00210=513669
BC00211=494109
BC00212=467540
BC00213=467540
BC00214=478876
BC00215=478876
BC00216=478876
BC00217=478876
BC00218=478876
BC00219=478876
BC00220=478876
BC00221=478876
BC00222=478876
BC00223=478876
BC00224=478876
BC00225=478876
BC00226=481980
BC00227=563952
BC00228=606256
BC00229=606256
BC00230=606252
BC00231=606252
BC00232=606252
BC00233=654662
BC00234=654618
BC00235=654618
BC00236=654618
BC00237=654618
BC00238=654618
BC00239=654618
BC00240=654618
BC00241=654618
BC00242=686402
BC00243=686402
BC00244=686402
BC00245=686402
BC00246=652574
BC00247=641414
BC00248=715810
BC00249=784046
BC00250=784046
BC00251=784046
BC00252=784046
BC00253=784046
BC00254=784046
BC00255=784046
BC00256=784043
BC00257=784043
BC00258=784046
BC00259=821134
BC00260=821134
BC00261=821134
BC00262=821134
BC00263=821134
BC00264=821134
BC00265=821134
BC00266=821134
BC00267=821134
BC00268=821134
BC00269=821133
BC00270=821133
BC00271=821134
BC00272=851941
BC00273=859414
BC00274=859414
BC00275=859414
BC00276=859414
BC00277=876203
BC00278=876203
BC00279=876203
BC00280=909600
BC00281=945583
BC00282=1005127
BC00283=999652
BC00284=999652
BC00285=991093
BC00286=990930
BC00287=990930
BC00288=990930
BC00289=990930
BC00290=990930
BC00291=990930
BC00292=990930
BC00293=981572
BC00294=972138
BC00295=892453
BC00296=828403
BC00297=518986
BC00298=509920
BC00299=467540
BC00300=467540
BC00301=467540
BC00302=521167
BC00303=520352
BC00304=535759
BC00305=535759
BC00306=535757
BC00307=535757
BC00308=535757
BC00309=535757
BC00310=485653
BC00311=485653
BC00312=485653
BC00313=485653
BC00314=485653
BC00315=485653
BC00316=485655
BC00317=485655
BC00318=485653
BC00319=485653
BC00320=485653
BC00321=615112
BC00322=615112
BC00323=615112
BC00324=615112
BC00325=615112
BC00326=615112
BC00327=615112
BC00328=615112
BC00329=615112
BC00330=615112
BC00331=615112
BC00332=615112
BC00333=615112
BC00334=615112
BC00335=615112
BC00336=658076
BC00337=658076
BC00338=658076
BC00339=658076
BC00340=655680
BC00341=643721
BC00342=643721
BC00343=793396
BC00344=799070
BC00345=799070
BC00346=799070
BC00347=799070
BC00348=799070
BC00349=799070
BC00350=799070
BC00351=799070
BC00352=799070
BC00353=799070
BC00354=799070
BC00355=799070
BC00356=799070
BC00357=845667
BC00358=845667
BC00359=845667
BC00360=845667
BC00361=845667
BC00362=845667
BC00363=845667
BC00364=845667
BC00365=845667
BC00366=845667
BC00367=845667
BC00368=845667
BC00369=874192
BC00370=874192
BC00371=874192
BC00372=874192
BC00373=891286
BC00374=862979
BC00375=977267
BC00376=1008066
BC00377=1008066
BC00378=995068
BC00379=995068
BC00380=995068
BC00381=1008066
BC00382=1008066
BC00383=1008066
BC00384=1008066
BC00385=895479
BC00386=639407
BC00387=467225
BC00388=513669
BC00389=542621
BC00390=535309
BC00391=478364
BC00392=478364
BC00393=478876
BC00394=466587
BC00395=466587
BC00396=466587
BC00397=466587
BC00398=471196
BC00399=471196
BC00400=471196
BC00401=471196
BC00402=471196
BC00403=463516
BC00404=463516
BC00405=463516
BC00406=463516
BC00407=463516
BC00408=478876
BC00409=480759
BC00410=480759
BC00411=560395
BC00412=606256
BC00413=606256
BC00414=606252
BC00415=606252
BC00416=606252
BC00417=606252
BC00418=654662
BC00419=654618
BC00420=654618
BC00421=654618
BC00422=654618
BC00423=654618
BC00424=646938
BC00425=646938
BC00426=646938
BC00427=646938
BC00428=646938
BC00429=674113
BC00430=674113
BC00431=674061
BC00432=674061
BC00433=674113
BC00434=652574
BC00435=652574
BC00436=774850
BC00437=784046
BC00438=784046
BC00439=768685
BC00440=768685
BC00441=768685
BC00442=768685
BC00443=753324
BC00444=753324
BC00445=753324
BC00446=753324
BC00447=753324
BC00448=782732
BC00449=782732
BC00450=782732
BC00451=782732
BC00452=782732
BC00453=778123
BC00454=778123
BC00455=778123
BC00456=778123
BC00457=778123
BC00458=816525
BC00459=816525
BC00460=816525
BC00461=816525
BC00462=816525
BC00463=854928
BC00464=854928
BC00465=854928
BC00466=854928
BC00467=854928
BC00468=893330
BC00469=893330
BC00470=893330
BC00471=893330
BC00472=893330
BC00473=909600
BC00474=995060
BC00475=999652
BC00476=999652
BC00477=1006454
BC00478=1006291
BC00479=1006291
BC00480=1006291
BC00481=1006291
BC00482=998610
BC00483=998610
BC00484=998610
BC00485=998610
BC00486=998610
BC00487=981572
BC00488=972138
BC00489=828403
BC00490=518986
BC00491=509920
BC00492=467540
BC00493=497868
BC00494=497868
BC00495=535759
BC00496=535759
BC00497=528077
BC00498=528077
BC00499=528077
BC00500=528077
BC00501=535757
BC00502=485653
BC00503=477973
BC00504=477973
BC00505=477973
BC00506=477973
BC00507=477973
BC00508=485653
BC00509=470292
BC00510=470292
BC00511=470292
BC00512=470292
BC00513=485653
BC00514=485653
BC00515=485653
BC00516=601945
BC00517=615112
BC00518=615112
BC00519=615112
BC00520=621256
BC00521=621256
BC00522=621256
BC00523=621256
BC00524=615112
BC00525=615112
BC00526=615112
BC00527=615112
BC00528=615112
BC00529=615112
BC00530=615112
BC00531=615112
BC00532=615112
BC00533=615112
BC00534=645787
BC00535=645787
BC00536=645787
BC00537=645787
BC00538=645787
BC00539=655680
BC00540=655680
BC00541=765678
BC00542=799070
BC00543=799070
BC00544=776029
BC00545=776029
BC00546=776029
BC00547=776029
BC00548=768348
BC00549=768348
BC00550=768348
BC00551=768348
BC00552=768348
BC00553=768348
BC00554=760668
BC00555=760668
BC00556=760668
BC00557=760668
BC00558=802656
BC00559=802656
BC00560=802656
BC00561=802656
BC00562=802656
BC00563=839522
BC00564=839522
BC00565=839522
BC00566=839522
BC00567=839522
BC00568=877924
BC00569=877924
BC00570=877924
BC00571=877924
BC00572=877924
BC00573=916326
BC00574=916326
BC00575=916326
BC00576=916326
BC00577=916326
BC00578=899436
BC00579=943124
BC00580=971560
BC00581=1008066
BC00582=1008066
BC00583=1005821
BC00584=1005821
BC00585=1005821
BC00586=1005821
BC00587=1015746
BC00588=1015746
BC00589=1015746
BC00590=1015746
BC00591=1008066
BC00592=895479
BC00593=639407
BC00594=467225
BC00595=513669
BC00596=494109
BC00597=467540
BC00598=467540
BC00599=478876
BC00600=477344
BC00601=469580
BC00602=478876
BC00603=469940
BC00604=469940
BC00605=478876
BC00606=478876
BC00607=478876
BC00608=478876
BC00609=478876
BC00610=478876
BC00611=479530
BC00612=502776
BC00613=571156
BC00614=606256
BC00615=606256
BC00616=606252
BC00617=606252
BC00618=606252
BC00619=654662
BC00620=654618
BC00621=654618
BC00622=654618
BC00623=654618
BC00624=654618
BC00625=654618
BC00626=654618
BC00627=654618
BC00628=686402
BC00629=686402
BC00630=686402
BC00631=686402
BC00632=652574
BC00633=654591
BC00634=763025
BC00635=784046
BC00636=784046
BC00637=784046
BC00638=784046
BC00639=784046
BC00640=784046
BC00641=784043
BC00642=784043
BC00643=784046
BC00644=821134
BC00645=821134
BC00646=821134
BC00647=821134
BC00648=821134
BC00649=821134
BC00650=821134
BC00651=821134
BC00652=859536
BC00653=859536
BC00654=859536
BC00655=859536
BC00656=897938
BC00657=897938
BC00658=897938
BC00659=897938
BC00660=936340
BC00661=936340
BC00662=936340
BC00663=936340
BC00664=909600
BC00665=909600
BC00666=972020
BC00667=999652
BC00668=999652
BC00669=991093
BC00670=990930
BC00671=990930
BC00672=990930
BC00673=990930
BC00674=990930
BC00675=990930
BC00676=990930
BC00677=981572
BC00678=972138
BC00679=920868
BC00680=828403
BC00681=518986
BC00682=509920
BC00683=467540
BC00684=467540
BC00685=467540
BC00686=521167
BC00687=520352
BC00688=535759
BC00689=535759
BC00690=535757
BC00691=535757
BC00692=535757
BC00693=535757
BC00694=485653
BC00695=485653
BC00696=485653
BC00697=485653
BC00698=485653
BC00699=485653
BC00700=485653
BC00701=485653
BC00702=485653
BC00703=485653
BC00704=485653
BC00705=600333
BC00706=615112
BC00707=615112
BC00708=615112
BC00709=615112
BC00710=615112
BC00711=615112
BC00712=615112
BC00713=615112
BC00714=615112
BC00715=615112
BC00716=615112
BC00717=615112
BC00718=615112
BC00719=615112
BC00720=658076
BC00721=658076
BC00722=658076
BC00723=658076
BC00724=655680
BC00725=656245
BC00726=762546
BC00727=762546
BC00728=799070
BC00729=799070
BC00730=799068
BC00731=799068
BC00732=799070
BC00733=799070
BC00734=799070
BC00735=799070
BC00736=799070
BC00737=799070
BC00738=799070
BC00739=799070
BC00740=799070
BC00741=845667
BC00742=845667
BC00743=845667
BC00744=845667
BC00745=884069
BC00746=884069
BC00747=884069
BC00748=884069
BC00749=922471
BC00750=922471
BC00751=922471
BC00752=922471
BC00753=960873
BC00754=960873
BC00755=960873
BC00756=947507
BC00757=899436
BC00758=899436
BC00759=981307
BC00760=1008066
BC00761=997960
BC00762=997960
BC00763=1008527
BC00764=1008527
BC00765=995068
BC00766=1008066
BC00767=1008066
BC00768=1008066
BC00769=1008066
BC00770=1008066
BC00771=895479
BC00772=639407
///POSTYPE BASE
///RECTAN
///RCONF 0,0,0,0,0,0,0,0,0,0,0,0,0,0,0,0,0,0,0,0,0,0,0,0
P00006=-2.449,0.031,8.825,0.0000,0.0000,0.0000
P00056=0.000,0.000,5.000,0.0000,0.0000,0.0000
P00301=0.005,-4.708,-4.628,0.0000,0.0000,0.0000
P00302=0.052,-2.937,-4.426,0.0000,0.0000,0.0000
P00303=-0.004,-1.437,-4.584,0.0000,0.0000,0.0000
P00304=0.028,-1.666,-4.234,0.0000,0.0000,0.0000
P00305=-0.003,-1.920,-3.501,0.0000,0.0000,0.0000
P00306=0.015,-2.252,-3.054,0.0000,0.0000,0.0000
P00307=0.019,-2.151,-5.077,0.0000,0.0000,0.0000
P00308=-0.003,-2.092,-4.888,0.0000,0.0000,0.0000
P00309=-0.040,-2.205,-4.992,0.0000,0.0000,0.0000
P00310=-0.006,-2.490,-5.925,0.0000,0.0000,0.0000
P00311=-0.007,-2.079,-5.307,0.0000,0.0000,0.0000
P00312=-0.032,2.202,-7.632,0.0000,0.0000,0.0000
///RCONF 1,0,0,0,0,0,0,0,0,0,0,0,0,0,0,0,0,0,0,0,0,0,0,0
P00313=-0.088,1.055,2.110,0.0000,0.0000,0.0000
P00314=-0.055,1.752,1.634,0.0000,0.0000,0.0000
P00315=-0.074,0.897,1.645,0.0000,0.0000,0.0000
P00316=0.009,2.112,2.075,0.0000,0.0000,0.0000
///RCONF 0,0,0,0,0,0,0,0,0,0,0,0,0,0,0,0,0,0,0,0,0,0,0,0
P00351=13.563,-0.027,-0.653,0.0000,0.0000,0.0000
P00352=13.252,-0.027,-0.827,0.0000,0.0000,0.0000
P00353=10.971,-0.082,0.776,0.0000,0.0000,0.0000
P00354=-0.024,2.508,-1.824,0.0000,0.0000,0.0000
P00355=-0.001,2.528,-1.131,0.0000,0.0000,0.0000
P00356=-0.034,2.921,-0.262,0.0000,0.0000,0.0000
P00357=0.003,3.386,-0.091,0.0000,0.0000,0.0000
P00358=0.014,3.037,-0.020,0.0000,0.0000,0.0000
P00359=-0.005,2.731,0.912,0.0000,0.0000,0.0000
P00360=-0.011,3.412,0.438,0.0000,0.0000,0.0000
P00361=0.018,3.050,1.253,0.0000,0.0000,0.0000
P00362=0.014,2.784,0.148,0.0000,0.0000,0.0000
P00363=0.026,4.310,-2.639,0.0000,0.0000,0.0000
P00364=0.034,4.181,-4.040,0.0000,0.0000,0.0000
P00365=-0.020,3.204,-1.693,0.0000,0.0000,0.0000
P00366=0.018,3.878,-1.790,0.0000,0.0000,0.0000
//INST
///DATE 2025/06/05 10:41
///ATTR SC,RW
///GROUP1 RB1,BS1
NOP
CALL JOB:MOVE_INTO_TUNNEL
MOVJ C00000 BC00000 VJ=10.00
MOVJ C00001 BC00001 VJ=10.00
MOVJ C00002 BC00002 VJ=10.00
MOVJ C00003 BC00003 VJ=10.00
MOVJ C00004 BC00004 VJ=10.00
'------------------------
'W29.2
'------------------------
MOVL C00005 BC00005 V=500.0
'------------------------
'W63.5
'------------------------
SFTOF
MOVL C00006 BC00006 V=166.7 PL=0
REFP 3 C00007 BC00007
CALL JOB:SEARCH-R1
IMOV P0056 V=50.0 PL=0
SET P0301 P0006
SFTON P0301
REFP 3 C00008 BC00008
CALL JOB:SEARCH-R1
SET P0301 P0006
SFTON P0301
MOVL C00009 BC00009 V=166.7 PL=0
SFTOF
MOVL C00010 BC00010 V=500.0
MOVL C00011 BC00011 V=166.7 PL=0
REFP 3 C00012 BC00012
CALL JOB:SEARCH-R1
IMOV P0056 V=50.0 PL=0
SET P0302 P0006
SFTON P0302
REFP 3 C00013 BC00013
CALL JOB:SEARCH-R1
SET P0302 P0006
SFTON P0302
MOVL C00014 BC00014 V=166.7 PL=0
SFTOF
MOVL C00015 BC00015 V=500.0
MOVL C00016 BC00016 V=166.7 PL=0
REFP 3 C00017 BC00017
CALL JOB:SEARCH-R1
IMOV P0056 V=50.0 PL=0
SET P0303 P0006
SFTON P0303
REFP 3 C00018 BC00018
CALL JOB:SEARCH-R1
SET P0303 P0006
SFTON P0303
SFTOF
MOVL C00019 BC00019 V=166.7 PL=0
MOVL C00020 BC00020 V=500.0
MOVJ C00021 BC00021 VJ=30.00
MOVJ C00022 BC00022 VJ=30.00
MOVJ C00023 BC00023 VJ=30.00
MOVL C00024 BC00024 V=500.0
'------------------------
'W29.14
'------------------------
MOVL C00025 BC00025 V=166.7 PL=0
REFP 3 C00026 BC00026
CALL JOB:SEARCH-R1
IMOV P0056 V=23.0 PL=0
SET P0304 P0006
SFTON P0304
REFP 3 C00027 BC00027
CALL JOB:SEARCH-R1
SET P0304 P0006
SFTON P0304
MOVL C00028 BC00028 V=66.7 PL=0
SFTOF
'PRZEJAZD
MOVL C00029 BC00029 V=500.0
MOVL C00030 BC00030 V=500.0
'------------------------
'W63.17
'------------------------
MOVL C00031 BC00031 V=166.7 PL=0
REFP 3 C00032 BC00032
CALL JOB:SEARCH-R1
IMOV P0056 V=23.0 PL=0
SET P0305 P0006
SFTON P0305
REFP 3 C00033 BC00033
CALL JOB:SEARCH-R1
SET P0305 P0006
SFTON P0305
MOVL C00034 BC00034 V=166.7 PL=0
SFTOF
MOVL C00035 BC00035 V=500.0
MOVL C00036 BC00036 V=166.7
REFP 3 C00037 BC00037
CALL JOB:SEARCH-R1
IMOV P0056 V=23.0 PL=0
SET P0306 P0006
SFTON P0306
REFP 3 C00038 BC00038
CALL JOB:SEARCH-R1
SET P0306 P0006
SFTON P0306
MOVL C00039 BC00039 V=166.7 PL=0
'PRZEJAZD
MOVL C00040 BC00040 V=500.0
MOVL C00041 BC00041 V=166.7
REFP 3 C00042 BC00042
CALL JOB:SEARCH-R1
IMOV P0056 V=23.0 PL=0
SET P0307 P0006
SFTON P0307
REFP 3 C00043 BC00043
CALL JOB:SEARCH-R1
SET P0307 P0006
SFTON P0307
MOVL C00044 BC00044 V=166.7 PL=0
SFTOF
MOVJ C00045 BC00045 VJ=20.00
MOVJ C00046 BC00046 VJ=20.00
MOVJ C00047 BC00047 VJ=30.00
MOVJ C00048 BC00048 VJ=30.00
MOVJ C00049 BC00049 VJ=30.00
MOVL C00050 BC00050 V=500.0
'------------------------
'W63.20
'------------------------
MOVL C00051 BC00051 V=166.7 PL=0
REFP 3 C00052 BC00052
CALL JOB:SEARCH-R1
IMOV P0056 V=23.0 PL=0
SET P0308 P0006
SFTON P0308
REFP 3 C00053 BC00053
CALL JOB:SEARCH-R1
SET P0308 P0006
SFTON P0308
MOVL C00054 BC00054 V=166.7 PL=0
SFTOF
'PRZEJAZD
MOVL C00055 BC00055 V=500.0
'------------------------
'W63.23
'------------------------
MOVL C00056 BC00056 V=166.7 PL=0
REFP 3 C00057 BC00057
CALL JOB:SEARCH-R1
IMOV P0056 V=23.0 PL=0
SET P0309 P0006
SFTON P0309
REFP 3 C00058 BC00058
CALL JOB:SEARCH-R1
SET P0309 P0006
SFTON P0309
MOVL C00059 BC00059 V=250.0 PL=0
SFTOF
MOVL C00060 BC00060 V=500.0
MOVL C00061 BC00061 V=166.7 PL=0
REFP 3 C00062 BC00062
CALL JOB:SEARCH-R1
IMOV P0056 V=23.0 PL=0
SET P0310 P0006
SFTON P0310
REFP 3 C00063 BC00063
CALL JOB:SEARCH-R1
SET P0310 P0006
SFTON P0310
MOVL C00064 BC00064 V=250.0 PL=0
SFTOF
MOVL C00065 BC00065 V=500.0
MOVL C00066 BC00066 V=166.7 PL=0
REFP 3 C00067 BC00067
CALL JOB:SEARCH-R1
IMOV P0056 V=23.0 PL=0
SET P0311 P0006
SFTON P0311
REFP 3 C00068 BC00068
CALL JOB:SEARCH-R1
SET P0311 P0006
SFTON P0311
MOVL C00069 BC00069 V=250.0 PL=0
SFTOF
MOVL C00070 BC00070 V=500.0
MOVL C00071 BC00071 V=166.7 PL=0
REFP 3 C00072 BC00072
CALL JOB:SEARCH-R1
IMOV P0056 V=23.0 PL=0
SET P0312 P0006
SFTON P0312
REFP 3 C00073 BC00073
CALL JOB:SEARCH-R1
SET P0312 P0006
SFTON P0312
MOVL C00074 BC00074 V=250.0 PL=0
SFTOF
MOVL C00075 BC00075 V=333.3
'------------------------
'W29.29
'------------------------
MOVL C00076 BC00076 V=166.7 PL=0
REFP 3 C00077 BC00077
CALL JOB:SEARCH-R1
IMOV P0056 V=23.0 PL=0
SET P0313 P0006
SFTON P0313
REFP 3 C00078 BC00078
CALL JOB:SEARCH-R1
SET P0313 P0006
SFTON P0313
MOVL C00079 BC00079 V=250.0 PL=0
SFTOF
MOVL C00080 BC00080 V=333.3
'------------------------
'W29.29
'------------------------
MOVL C00081 BC00081 V=166.7 PL=0
REFP 3 C00082 BC00082
CALL JOB:SEARCH-R1
IMOV P0056 V=23.0 PL=0
SET P0314 P0006
SFTON P0314
REFP 3 C00083 BC00083
CALL JOB:SEARCH-R1
SET P0314 P0006
SFTON P0314
MOVL C00084 BC00084 V=250.0 PL=0
SFTOF
'PRZEJAZD
MOVL C00085 BC00085 V=333.3
'PRZEJAZD
MOVL C00086 BC00086 V=500.0
MOVL C00087 BC00087 V=500.0
MOVL C00088 BC00088 V=333.3
MOVL C00089 BC00089 V=333.3
MOVL C00090 BC00090 V=166.7 PL=0
REFP 3 C00091 BC00091
CALL JOB:SEARCH-R1
IMOV P0056 V=23.0 PL=0
SET P0315 P0006
SFTON P0315
REFP 3 C00092 BC00092
CALL JOB:SEARCH-R1
SET P0315 P0006
SFTON P0315
MOVL C00093 BC00093 V=250.0 PL=0
SFTOF
MOVL C00094 BC00094 V=333.3
MOVL C00095 BC00095 V=166.7 PL=0
REFP 3 C00096 BC00096
CALL JOB:SEARCH-R1
IMOV P0056 V=23.0 PL=0
SET P0316 P0006
SFTON P0316
REFP 3 C00097 BC00097
CALL JOB:SEARCH-R1
SET P0316 P0006
SFTON P0316
MOVL C00098 BC00098 V=250.0 PL=0
SFTOF
MOVJ C00099 BC00099 VJ=10.00
MOVJ C00100 BC00100 VJ=10.00
MOVJ C00101 BC00101 VJ=30.00
MOVJ C00102 BC00102 VJ=20.00
MOVJ C00103 BC00103 VJ=50.00
MOVJ C00104 BC00104 VJ=20.00
MOVJ C00105 BC00105 VJ=10.00
MOVJ C00106 BC00106 VJ=20.00
MOVJ C00107 BC00107 VJ=20.00
'------------------------
'W28.2
'------------------------
MOVJ C00108 BC00108 VJ=10.00
MOVJ C00109 BC00109 VJ=10.00
MOVL C00110 BC00110 V=500.0
MOVL C00111 BC00111 V=500.0
'------------------------
'W62.5
'------------------------
MOVL C00112 BC00112 V=166.7 PL=0
REFP 3 C00113 BC00113
CALL JOB:SEARCH-R1
IMOV P0056 V=23.0 PL=0
SET P0351 P0006
SFTON P0351
REFP 3 C00114 BC00114
CALL JOB:SEARCH-R1
SET P0351 P0006
SFTON P0351
MOVL C00115 BC00115 V=250.0 PL=0
SFTOF
'PRZEJAZD
MOVL C00116 BC00116 V=500.0
MOVL C00117 BC00117 V=500.0
MOVL C00118 BC00118 V=500.0
MOVL C00119 BC00119 V=166.7 PL=0
REFP 3 C00120 BC00120
CALL JOB:SEARCH-R1
IMOV P0056 V=23.0 PL=0
SET P0352 P0006
SFTON P0352
REFP 3 C00121 BC00121
CALL JOB:SEARCH-R1
SET P0352 P0006
SFTON P0352
MOVL C00122 BC00122 V=250.0 PL=0
SFTOF
MOVL C00123 BC00123 V=500.0
'------------------------
'W29.8
'------------------------
MOVL C00124 BC00124 V=166.7 PL=0
REFP 3 C00125 BC00125
CALL JOB:SEARCH-R1
IMOV P0056 V=23.0 PL=0
SET P0353 P0006
SFTON P0353
REFP 3 C00126 BC00126
CALL JOB:SEARCH-R1
SET P0353 P0006
SFTON P0353
MOVL C00127 BC00127 V=250.0 PL=0
SFTOF
MOVL C00128 BC00128 V=500.0
'PRZEJAZD
MOVL C00129 BC00129 V=500.0
MOVJ C00130 BC00130 VJ=20.00
MOVL C00131 BC00131 V=500.0
MOVL C00132 BC00132 V=500.0
MOVL C00133 BC00133 V=500.0
'------------------------
'W29.11
'------------------------
MOVL C00134 BC00134 V=166.7 PL=0
REFP 3 C00135 BC00135
CALL JOB:SEARCH-R1
IMOV P0056 V=23.0 PL=0
SET P0354 P0006
SFTON P0354
REFP 3 C00136 BC00136
CALL JOB:SEARCH-R1
SET P0354 P0006
SFTON P0354
MOVL C00137 BC00137 V=250.0 PL=0
SFTOF
'PRZEJAZD
MOVL C00138 BC00138 V=500.0
'------------------------
'W29.14
'------------------------
MOVL C00139 BC00139 V=166.7 PL=0
REFP 3 C00140 BC00140
CALL JOB:SEARCH-R1
IMOV P0056 V=23.0 PL=0
SET P0355 P0006
SFTON P0355
REFP 3 C00141 BC00141
CALL JOB:SEARCH-R1
SET P0355 P0006
SFTON P0355
MOVL C00142 BC00142 V=250.0 PL=0
SFTOF
'PRZEJAZD
MOVL C00143 BC00143 V=500.0
'------------------------
'W63.17
'------------------------
MOVL C00144 BC00144 V=166.7 PL=0
REFP 3 C00145 BC00145
CALL JOB:SEARCH-R1
IMOV P0056 V=23.0 PL=0
SET P0356 P0006
SFTON P0356
REFP 3 C00146 BC00146
CALL JOB:SEARCH-R1
SET P0356 P0006
SFTON P0356
MOVL C00147 BC00147 V=250.0 PL=0
SFTOF
MOVL C00148 BC00148 V=500.0
MOVL C00149 BC00149 V=166.7 PL=0
REFP 3 C00150 BC00150
CALL JOB:SEARCH-R1
IMOV P0056 V=23.0 PL=0
SET P0357 P0006
SFTON P0357
REFP 3 C00151 BC00151
CALL JOB:SEARCH-R1
SET P0357 P0006
SFTON P0357
MOVL C00152 BC00152 V=250.0 PL=0
SFTOF
'PRZEJAZD
MOVL C00153 BC00153 V=500.0
MOVJ C00154 BC00154 VJ=30.00
MOVJ C00155 BC00155 VJ=30.00
MOVJ C00156 BC00156 VJ=30.00
MOVL C00157 BC00157 V=500.0
MOVL C00158 BC00158 V=500.0
'------------------------
'W62.20
'------------------------
MOVL C00159 BC00159 V=166.7 PL=0
REFP 3 C00160 BC00160
CALL JOB:SEARCH-R1
IMOV P0056 V=23.0 PL=0
SET P0358 P0006
SFTON P0358
REFP 3 C00161 BC00161
CALL JOB:SEARCH-R1
SET P0358 P0006
SFTON P0358
MOVL C00162 BC00162 V=250.0 PL=0
SFTOF
'PRZEJAZD
MOVL C00163 BC00163 V=500.0
'------------------------
'W63.23
'------------------------
MOVL C00164 BC00164 V=166.7 PL=0
REFP 3 C00165 BC00165
CALL JOB:SEARCH-R1
IMOV P0056 V=23.0 PL=0
SET P0359 P0006
SFTON P0359
REFP 3 C00166 BC00166
CALL JOB:SEARCH-R1
SET P0359 P0006
SFTON P0359
MOVL C00167 BC00167 V=250.0 PL=0
SFTOF
MOVL C00168 BC00168 V=500.0
'------------------------
'W29.29
'------------------------
MOVL C00169 BC00169 V=166.7 PL=0
REFP 3 C00170 BC00170
CALL JOB:SEARCH-R1
IMOV P0056 V=23.0 PL=0
SET P0360 P0006
SFTON P0360
REFP 3 C00171 BC00171
CALL JOB:SEARCH-R1
SET P0360 P0006
SFTON P0360
MOVL C00172 BC00172 V=250.0 PL=0
SFTOF
'PRZEJAZD
MOVL C00173 BC00173 V=500.0
MOVL C00174 BC00174 V=166.7 PL=0
REFP 3 C00175 BC00175
CALL JOB:SEARCH-R1
IMOV P0056 V=23.0 PL=0
SET P0361 P0006
SFTON P0361
REFP 3 C00176 BC00176
CALL JOB:SEARCH-R1
SET P0361 P0006
SFTON P0361
MOVL C00177 BC00177 V=250.0 PL=0
SFTOF
MOVL C00178 BC00178 V=500.0
MOVL C00179 BC00179 V=166.7 PL=0
REFP 3 C00180 BC00180
CALL JOB:SEARCH-R1
IMOV P0056 V=23.0 PL=0
SET P0362 P0006
SFTON P0362
REFP 3 C00181 BC00181
CALL JOB:SEARCH-R1
SET P0362 P0006
SFTON P0362
MOVL C00182 BC00182 V=250.0 PL=0
SFTOF
MOVL C00183 BC00183 V=500.0
MOVL C00184 BC00184 V=166.7 PL=0
REFP 3 C00185 BC00185
CALL JOB:SEARCH-R1
IMOV P0056 V=23.0 PL=0
SET P0363 P0006
SFTON P0363
REFP 3 C00186 BC00186
CALL JOB:SEARCH-R1
SET P0363 P0006
SFTON P0363
MOVL C00187 BC00187 V=250.0 PL=0
SFTOF
MOVL C00188 BC00188 V=500.0
MOVL C00189 BC00189 V=166.7 PL=0
REFP 3 C00190 BC00190
CALL JOB:SEARCH-R1
IMOV P0056 V=23.0 PL=0
SET P0364 P0006
SFTON P0364
REFP 3 C00191 BC00191
CALL JOB:SEARCH-R1
SET P0364 P0006
SFTON P0364
MOVL C00192 BC00192 V=250.0 PL=0
SFTOF
'------------------------
'W29.32
'------------------------
'PRZEJAZD
MOVL C00193 BC00193 V=500.0
MOVJ C00194 BC00194 VJ=30.00
MOVJ C00195 BC00195 VJ=15.00
MOVJ C00196 BC00196 VJ=15.00
MOVL C00197 BC00197 V=166.7
MOVL C00198 BC00198 V=166.7 PL=0
REFP 3 C00199 BC00199
CALL JOB:SEARCH-R1
IMOV P0056 V=23.0 PL=0
SET P0365 P0006
SFTON P0365
REFP 3 C00200 BC00200
CALL JOB:SEARCH-R1
SET P0365 P0006
SFTON P0365
MOVL C00201 BC00201 V=250.0 PL=0
SFTOF
MOVL C00202 BC00202 V=166.7 PL=0
REFP 3 C00203 BC00203
CALL JOB:SEARCH-R1
IMOV P0056 V=23.0 PL=0
SET P0366 P0006
SFTON P0366
REFP 3 C00204 BC00204
CALL JOB:SEARCH-R1
SET P0366 P0006
SFTON P0366
MOVL C00205 BC00205 V=250.0 PL=0
SFTOF
MOVJ C00206 BC00206 VJ=20.00
MOVJ C00207 BC00207 VJ=30.00
MOVJ C00208 BC00208 VJ=30.00
'KONIEC SEARCH WEW STRONA
MOVJ C00209 BC00209 VJ=30.00
MOVJ C00210 BC00210 VJ=20.00
MOVJ C00211 BC00211 VJ=10.00
MOVJ C00212 BC00212 VJ=20.00
MOVJ C00213 BC00213 VJ=20.00
'------------------------
'W29.2
'------------------------
MOVL C00214 BC00214 V=500.0
'------------------------
'W63.5
MACRO1 MJ#(0) ARGF9
'------------------------
SFTOF
SFTON P0301
MOVL C00215 BC00215 V=166.7 PL=0
ARCON
MOVL C00216 BC00216 V=10.0
ARCOF
SFTOF
MOVL C00217 BC00217 V=500.0
SFTON P0302
MOVL C00218 BC00218 V=166.7 PL=0
ARCON
MOVL C00219 BC00219 V=10.0
ARCOF
MOVL C00220 BC00220 V=166.7 PL=0
SFTOF
MOVL C00221 BC00221 V=500.0
SFTON P0303
MOVL C00222 BC00222 V=166.7 PL=0
ARCON
MOVL C00223 BC00223 V=10.0
ARCOF
SFTOF
MOVL C00224 BC00224 V=166.7 PL=0
MOVL C00225 BC00225 V=500.0
MOVJ C00226 BC00226 VJ=30.00
MOVJ C00227 BC00227 VJ=30.00
MOVJ C00228 BC00228 VJ=30.00
MOVL C00229 BC00229 V=500.0
'------------------------
'W29.14
'------------------------
SFTON P0304
MOVL C00230 BC00230 V=166.7 PL=0
ARCON
MOVL C00231 BC00231 V=10.0
ARCOF
MOVL C00232 BC00232 V=166.7 PL=0
SFTOF
'PRZEJAZD
MOVL C00233 BC00233 V=500.0
MOVL C00234 BC00234 V=500.0
'------------------------
'W63.17
'------------------------
SFTON P0305
MOVL C00235 BC00235 V=166.7 PL=0
ARCON
MOVL C00236 BC00236 V=10.0
ARCOF
MOVL C00237 BC00237 V=166.7 PL=0
SFTOF
MOVL C00238 BC00238 V=500.0
SFTON P0306
MOVL C00239 BC00239 V=166.7
ARCON
MOVL C00240 BC00240 V=10.0
ARCOF
MOVL C00241 BC00241 V=166.7 PL=0
SFTOF
'PRZEJAZD
MOVL C00242 BC00242 V=500.0
SFTON P0307
MOVL C00243 BC00243 V=166.7
ARCON
MOVL C00244 BC00244 V=10.0
ARCOF
MOVL C00245 BC00245 V=166.7 PL=0
SFTOF
MOVJ C00246 BC00246 VJ=20.00
MOVJ C00247 BC00247 VJ=20.00
MOVJ C00248 BC00248 VJ=30.00
MOVJ C00249 BC00249 VJ=30.00
MOVJ C00250 BC00250 VJ=30.00
MOVL C00251 BC00251 V=500.0
'------------------------
'W63.20
'------------------------
SFTON P0308
MOVL C00252 BC00252 V=166.7 PL=0
ARCON
MOVL C00253 BC00253 V=10.0
ARCOF
MOVL C00254 BC00254 V=166.7 PL=0
SFTOF
'PRZEJAZD
MOVL C00255 BC00255 V=500.0
'------------------------
'W63.23
'------------------------
SFTON P0309
MOVL C00256 BC00256 V=166.7 PL=0
ARCON
MOVL C00257 BC00257 V=10.0
ARCOF
MOVL C00258 BC00258 V=250.0 PL=0
SFTOF
MOVL C00259 BC00259 V=500.0
SFTON P0310
MOVL C00260 BC00260 V=166.7 PL=0
ARCON
MOVL C00261 BC00261 V=10.0
ARCOF
MOVL C00262 BC00262 V=250.0 PL=0
SFTOF
MOVL C00263 BC00263 V=500.0
SFTON P0311
MOVL C00264 BC00264 V=166.7 PL=0
ARCON
MOVL C00265 BC00265 V=10.0
ARCOF
MOVL C00266 BC00266 V=250.0 PL=0
SFTOF
MOVL C00267 BC00267 V=500.0
MOVL C00268 BC00268 V=500.0
SFTON P0312
MOVL C00269 BC00269 V=166.7 PL=0
ARCON
MOVL C00270 BC00270 V=10.0
ARCOF
MOVL C00271 BC00271 V=250.0 PL=0
SFTOF
MOVL C00272 BC00272 V=500.0
SFTON P0313
MOVL C00273 BC00273 V=166.7 PL=0
ARCON
MOVL C00274 BC00274 V=10.0
ARCOF
MOVL C00275 BC00275 V=250.0 PL=0
SFTOF
MOVL C00276 BC00276 V=500.0
MOVL C00277 BC00277 V=333.3
'------------------------
'W29.29
'------------------------
SFTON P0314
MOVL C00278 BC00278 V=166.7 PL=0
ARCON
MOVL C00279 BC00279 V=10.0
ARCOF
MOVL C00280 BC00280 V=250.0 PL=0
SFTOF
'PRZEJAZD
MOVL C00281 BC00281 V=333.3
'PRZEJAZD
'KONIEC SPAWANIA CZESCI WSPOLNEJ
MOVL C00282 BC00282 V=500.0
MOVL C00283 BC00283 V=500.0
MOVL C00284 BC00284 V=333.3
MOVL C00285 BC00285 V=333.3
SFTON P0315
MOVL C00286 BC00286 V=166.7 PL=0
ARCON
MOVL C00287 BC00287 V=10.0
ARCOF
MOVL C00288 BC00288 V=250.0 PL=0
SFTOF
MOVL C00289 BC00289 V=333.3
SFTON P0316
MOVL C00290 BC00290 V=166.7 PL=0
ARCON
MOVL C00291 BC00291 V=10.0
ARCOF
MOVL C00292 BC00292 V=250.0 PL=0
SFTOF
MOVJ C00293 BC00293 VJ=10.00
MOVJ C00294 BC00294 VJ=10.00
MOVJ C00295 BC00295 VJ=30.00
MOVJ C00296 BC00296 VJ=20.00
MOVJ C00297 BC00297 VJ=50.00
MOVJ C00298 BC00298 VJ=20.00
MOVJ C00299 BC00299 VJ=10.00
MOVJ C00300 BC00300 VJ=20.00
MOVJ C00301 BC00301 VJ=20.00
'------------------------
'W28.2
'------------------------
MOVJ C00302 BC00302 VJ=10.00
MOVJ C00303 BC00303 VJ=10.00
MOVL C00304 BC00304 V=500.0
MOVL C00305 BC00305 V=500.0
'------------------------
'W62.5
'------------------------
SFTON P0351
MOVL C00306 BC00306 V=166.7 PL=0
ARCON
MOVL C00307 BC00307 V=10.0
ARCOF
MOVL C00308 BC00308 V=250.0 PL=0
SFTOF
'PRZEJAZD
MOVL C00309 BC00309 V=500.0
MOVL C00310 BC00310 V=500.0
MOVL C00311 BC00311 V=500.0
SFTON P0352
MOVL C00312 BC00312 V=166.7 PL=0
ARCON
MOVL C00313 BC00313 V=10.0
ARCOF
MOVL C00314 BC00314 V=250.0 PL=0
SFTOF
MOVL C00315 BC00315 V=500.0
'------------------------
'W29.8
'------------------------
SFTON P0353
MOVL C00316 BC00316 V=166.7 PL=0
ARCON
MOVL C00317 BC00317 V=10.0
ARCOF
MOVL C00318 BC00318 V=250.0 PL=0
SFTOF
MOVL C00319 BC00319 V=500.0
'PRZEJAZD
MOVL C00320 BC00320 V=500.0
MOVJ C00321 BC00321 VJ=20.00
MOVL C00322 BC00322 V=500.0
MOVL C00323 BC00323 V=500.0
MOVL C00324 BC00324 V=500.0
'------------------------
'W29.11
'------------------------
SFTON P0354
MOVL C00325 BC00325 V=166.7 PL=0
ARCON
MOVL C00326 BC00326 V=10.0
ARCOF
MOVL C00327 BC00327 V=250.0 PL=0
SFTOF
'PRZEJAZD
MOVL C00328 BC00328 V=500.0
'------------------------
'W29.14
'------------------------
SFTON P0355
MOVL C00329 BC00329 V=166.7 PL=0
ARCON
MOVL C00330 BC00330 V=10.0
ARCOF
MOVL C00331 BC00331 V=250.0 PL=0
SFTOF
'PRZEJAZD
MOVL C00332 BC00332 V=500.0
'------------------------
'W63.17
'------------------------
SFTON P0356
MOVL C00333 BC00333 V=166.7 PL=0
ARCON
MOVL C00334 BC00334 V=10.0
ARCOF
MOVL C00335 BC00335 V=250.0 PL=0
SFTOF
MOVL C00336 BC00336 V=500.0
SFTON P0357
MOVL C00337 BC00337 V=166.7 PL=0
ARCON
MOVL C00338 BC00338 V=10.0
ARCOF
MOVL C00339 BC00339 V=250.0 PL=0
SFTOF
'PRZEJAZD
MOVL C00340 BC00340 V=500.0
MOVJ C00341 BC00341 VJ=30.00
MOVJ C00342 BC00342 VJ=30.00
MOVJ C00343 BC00343 VJ=30.00
MOVL C00344 BC00344 V=500.0
MOVL C00345 BC00345 V=500.0
'------------------------
'W62.20
'------------------------
SFTON P0358
MOVL C00346 BC00346 V=166.7 PL=0
ARCON
MOVL C00347 BC00347 V=10.0
ARCOF
MOVL C00348 BC00348 V=250.0 PL=0
SFTOF
'PRZEJAZD
MOVL C00349 BC00349 V=500.0
'------------------------
'W63.23
'------------------------
SFTON P0359
MOVL C00350 BC00350 V=166.7 PL=0
ARCON
MOVL C00351 BC00351 V=10.0
ARCOF
MOVL C00352 BC00352 V=250.0 PL=0
MOVL C00353 BC00353 V=500.0
'------------------------
'W29.29
'------------------------
SFTON P0360
MOVL C00354 BC00354 V=166.7 PL=0
ARCON
MOVL C00355 BC00355 V=10.0
ARCOF
MOVL C00356 BC00356 V=250.0 PL=0
SFTOF
'PRZEJAZD
MOVL C00357 BC00357 V=500.0
SFTON P0361
MOVL C00358 BC00358 V=166.7 PL=0
ARCON
MOVL C00359 BC00359 V=10.0
ARCOF
MOVL C00360 BC00360 V=250.0 PL=0
SFTOF
MOVL C00361 BC00361 V=500.0
SFTON P0362
MOVL C00362 BC00362 V=166.7 PL=0
ARCON
MOVL C00363 BC00363 V=10.0
ARCOF
MOVL C00364 BC00364 V=250.0 PL=0
SFTOF
MOVL C00365 BC00365 V=500.0
SFTON P0363
MOVL C00366 BC00366 V=166.7 PL=0
ARCON
MOVL C00367 BC00367 V=10.0
ARCOF
MOVL C00368 BC00368 V=250.0 PL=0
SFTOF
'------------------------
'W29.32
'------------------------
'PRZEJAZD
MOVL C00369 BC00369 V=416.7
SFTON P0364
MOVL C00370 BC00370 V=166.7 PL=0
ARCON
MOVL C00371 BC00371 V=10.0
ARCOF
MOVL C00372 BC00372 V=250.0 PL=0
SFTOF
MOVJ C00373 BC00373 VJ=20.00
MOVJ C00374 BC00374 VJ=30.00
MOVJ C00375 BC00375 VJ=15.00
MOVJ C00376 BC00376 VJ=15.00
MOVL C00377 BC00377 V=166.7
SFTON P0365
MOVL C00378 BC00378 V=166.7 PL=0
ARCON
MOVL C00379 BC00379 V=10.0
ARCOF
MOVL C00380 BC00380 V=250.0 PL=0
SFTOF
SFTON P0366
MOVL C00381 BC00381 V=166.7 PL=0
ARCON
MOVL C00382 BC00382 V=10.0
ARCOF
MOVL C00383 BC00383 V=250.0 PL=0
SFTOF
MOVJ C00384 BC00384 VJ=20.00
MOVJ C00385 BC00385 VJ=30.00
MOVJ C00386 BC00386 VJ=30.00
CALL JOB:MOVE_OUT_OF_TUNNEL
CALL JOB:CLEAN-R1
CALL JOB:MOVE_INTO_TUNNEL
'KONIEC SPAWANIA WEW STRONA
MOVJ C00387 BC00387 VJ=10.00
MOVJ C00388 BC00388 VJ=10.00
MOVJ C00389 BC00389 VJ=20.00
MOVJ C00390 BC00390 VJ=20.00
MOVJ C00391 BC00391 VJ=10.00
MOVJ C00392 BC00392 VJ=10.00
'------------------------
'W29.2
'------------------------
MOVL C00393 BC00393 V=500.0
'------------------------
'W63.5
'------------------------
SFTOF
MOVL C00394 BC00394 V=166.7 PL=0
REFP 3 C00395 BC00395
CALL JOB:SEARCH-R1
IMOV P0056 V=50.0 PL=0
SET P0301 P0006
SFTON P0301
REFP 3 C00396 BC00396
CALL JOB:SEARCH-R1
SET P0301 P0006
SFTON P0301
MOVL C00397 BC00397 V=166.7 PL=0
SFTOF
MOVL C00398 BC00398 V=500.0
MOVL C00399 BC00399 V=166.7 PL=0
REFP 3 C00400 BC00400
CALL JOB:SEARCH-R1
IMOV P0056 V=50.0 PL=0
SET P0302 P0006
SFTON P0302
REFP 3 C00401 BC00401
CALL JOB:SEARCH-R1
SET P0302 P0006
SFTON P0302
MOVL C00402 BC00402 V=166.7 PL=0
SFTOF
MOVL C00403 BC00403 V=500.0
MOVL C00404 BC00404 V=166.7 PL=0
REFP 3 C00405 BC00405
CALL JOB:SEARCH-R1
IMOV P0056 V=50.0 PL=0
SET P0303 P0006
SFTON P0303
REFP 3 C00406 BC00406
CALL JOB:SEARCH-R1
SET P0303 P0006
SFTON P0303
SFTOF
MOVL C00407 BC00407 V=166.7 PL=0
MOVL C00408 BC00408 V=500.0
MOVJ C00409 BC00409 VJ=30.00
MOVJ C00410 BC00410 VJ=30.00
MOVJ C00411 BC00411 VJ=20.00
MOVJ C00412 BC00412 VJ=30.00
MOVL C00413 BC00413 V=500.0
'------------------------
'W29.14
'------------------------
MOVL C00414 BC00414 V=166.7 PL=0
REFP 3 C00415 BC00415
CALL JOB:SEARCH-R1
IMOV P0056 V=23.0 PL=0
SET P0304 P0006
SFTON P0304
REFP 3 C00416 BC00416
CALL JOB:SEARCH-R1
SET P0304 P0006
SFTON P0304
MOVL C00417 BC00417 V=66.7 PL=0
SFTOF
'PRZEJAZD
MOVL C00418 BC00418 V=500.0
MOVL C00419 BC00419 V=500.0
'------------------------
'W63.17
'------------------------
MOVL C00420 BC00420 V=166.7 PL=0
REFP 3 C00421 BC00421
CALL JOB:SEARCH-R1
IMOV P0056 V=23.0 PL=0
SET P0305 P0006
SFTON P0305
REFP 3 C00422 BC00422
CALL JOB:SEARCH-R1
SET P0305 P0006
SFTON P0305
MOVL C00423 BC00423 V=166.7 PL=0
SFTOF
MOVL C00424 BC00424 V=500.0
MOVL C00425 BC00425 V=166.7
REFP 3 C00426 BC00426
CALL JOB:SEARCH-R1
IMOV P0056 V=23.0 PL=0
SET P0306 P0006
SFTON P0306
REFP 3 C00427 BC00427
CALL JOB:SEARCH-R1
SET P0306 P0006
SFTON P0306
MOVL C00428 BC00428 V=166.7 PL=0
'PRZEJAZD
MOVL C00429 BC00429 V=500.0
MOVL C00430 BC00430 V=166.7
REFP 3 C00431 BC00431
CALL JOB:SEARCH-R1
IMOV P0056 V=23.0 PL=0
SET P0307 P0006
SFTON P0307
REFP 3 C00432 BC00432
CALL JOB:SEARCH-R1
SET P0307 P0006
SFTON P0307
MOVL C00433 BC00433 V=166.7 PL=0
SFTOF
MOVJ C00434 BC00434 VJ=20.00
MOVJ C00435 BC00435 VJ=20.00
MOVJ C00436 BC00436 VJ=30.00
MOVJ C00437 BC00437 VJ=30.00
MOVL C00438 BC00438 V=500.0
'------------------------
'W63.20
'------------------------
MOVL C00439 BC00439 V=166.7 PL=0
REFP 3 C00440 BC00440
CALL JOB:SEARCH-R1
IMOV P0056 V=23.0 PL=0
SET P0308 P0006
SFTON P0308
REFP 3 C00441 BC00441
CALL JOB:SEARCH-R1
SET P0308 P0006
SFTON P0308
MOVL C00442 BC00442 V=166.7 PL=0
SFTOF
'PRZEJAZD
MOVL C00443 BC00443 V=500.0
'------------------------
'W63.23
'------------------------
MOVL C00444 BC00444 V=166.7 PL=0
REFP 3 C00445 BC00445
CALL JOB:SEARCH-R1
IMOV P0056 V=23.0 PL=0
SET P0309 P0006
SFTON P0309
REFP 3 C00446 BC00446
CALL JOB:SEARCH-R1
SET P0309 P0006
SFTON P0309
MOVL C00447 BC00447 V=250.0 PL=0
SFTOF
MOVL C00448 BC00448 V=500.0
MOVL C00449 BC00449 V=166.7 PL=0
REFP 3 C00450 BC00450
CALL JOB:SEARCH-R1
IMOV P0056 V=23.0 PL=0
SET P0310 P0006
SFTON P0310
REFP 3 C00451 BC00451
CALL JOB:SEARCH-R1
SET P0310 P0006
SFTON P0310
MOVL C00452 BC00452 V=250.0 PL=0
SFTOF
MOVL C00453 BC00453 V=500.0
MOVL C00454 BC00454 V=166.7 PL=0
REFP 3 C00455 BC00455
CALL JOB:SEARCH-R1
IMOV P0056 V=23.0 PL=0
SET P0311 P0006
SFTON P0311
REFP 3 C00456 BC00456
CALL JOB:SEARCH-R1
SET P0311 P0006
SFTON P0311
MOVL C00457 BC00457 V=250.0 PL=0
SFTOF
MOVL C00458 BC00458 V=500.0
MOVL C00459 BC00459 V=166.7 PL=0
REFP 3 C00460 BC00460
CALL JOB:SEARCH-R1
IMOV P0056 V=23.0 PL=0
SET P0312 P0006
SFTON P0312
REFP 3 C00461 BC00461
CALL JOB:SEARCH-R1
SET P0312 P0006
SFTON P0312
MOVL C00462 BC00462 V=250.0 PL=0
SFTOF
MOVL C00463 BC00463 V=500.0
MOVL C00464 BC00464 V=166.7 PL=0
REFP 3 C00465 BC00465
CALL JOB:SEARCH-R1
IMOV P0056 V=23.0 PL=0
SET P0313 P0006
SFTON P0313
REFP 3 C00466 BC00466
CALL JOB:SEARCH-R1
SET P0313 P0006
SFTON P0313
MOVL C00467 BC00467 V=250.0 PL=0
SFTOF
MOVL C00468 BC00468 V=500.0
MOVL C00469 BC00469 V=166.7 PL=0
REFP 3 C00470 BC00470
CALL JOB:SEARCH-R1
IMOV P0056 V=23.0 PL=0
SET P0314 P0006
SFTON P0314
REFP 3 C00471 BC00471
CALL JOB:SEARCH-R1
SET P0314 P0006
SFTON P0314
MOVL C00472 BC00472 V=250.0 PL=0
SFTOF
'PRZEJAZD
MOVL C00473 BC00473 V=333.3
'PRZEJAZD
MOVL C00474 BC00474 V=500.0
MOVL C00475 BC00475 V=500.0
MOVL C00476 BC00476 V=333.3
MOVL C00477 BC00477 V=333.3
MOVL C00478 BC00478 V=166.7 PL=0
REFP 3 C00479 BC00479
CALL JOB:SEARCH-R1
IMOV P0056 V=23.0 PL=0
SET P0315 P0006
SFTON P0315
REFP 3 C00480 BC00480
CALL JOB:SEARCH-R1
SET P0315 P0006
SFTON P0315
MOVL C00481 BC00481 V=250.0 PL=0
SFTOF
MOVL C00482 BC00482 V=333.3
MOVL C00483 BC00483 V=166.7 PL=0
REFP 3 C00484 BC00484
CALL JOB:SEARCH-R1
IMOV P0056 V=23.0 PL=0
SET P0316 P0006
SFTON P0316
REFP 3 C00485 BC00485
CALL JOB:SEARCH-R1
SET P0316 P0006
SFTON P0316
MOVL C00486 BC00486 V=250.0 PL=0
SFTOF
MOVJ C00487 BC00487 VJ=10.00
MOVJ C00488 BC00488 VJ=10.00
MOVJ C00489 BC00489 VJ=20.00
MOVJ C00490 BC00490 VJ=50.00
MOVJ C00491 BC00491 VJ=20.00
MOVJ C00492 BC00492 VJ=10.00
'------------------------
'W28.2
'------------------------
MOVJ C00493 BC00493 VJ=10.00
MOVJ C00494 BC00494 VJ=10.00
MOVL C00495 BC00495 V=500.0
MOVL C00496 BC00496 V=500.0
'------------------------
'W62.5
'------------------------
MOVL C00497 BC00497 V=166.7 PL=0
REFP 3 C00498 BC00498
CALL JOB:SEARCH-R1
IMOV P0056 V=23.0 PL=0
SET P0351 P0006
SFTON P0351
REFP 3 C00499 BC00499
CALL JOB:SEARCH-R1
SET P0351 P0006
SFTON P0351
MOVL C00500 BC00500 V=250.0 PL=0
SFTOF
'PRZEJAZD
MOVL C00501 BC00501 V=500.0
MOVL C00502 BC00502 V=500.0
MOVL C00503 BC00503 V=500.0
MOVL C00504 BC00504 V=166.7 PL=0
REFP 3 C00505 BC00505
CALL JOB:SEARCH-R1
IMOV P0056 V=23.0 PL=0
SET P0352 P0006
SFTON P0352
REFP 3 C00506 BC00506
CALL JOB:SEARCH-R1
SET P0352 P0006
SFTON P0352
MOVL C00507 BC00507 V=250.0 PL=0
SFTOF
MOVL C00508 BC00508 V=500.0
'------------------------
'W29.8
'------------------------
MOVL C00509 BC00509 V=166.7 PL=0
REFP 3 C00510 BC00510
CALL JOB:SEARCH-R1
IMOV P0056 V=23.0 PL=0
SET P0353 P0006
SFTON P0353
REFP 3 C00511 BC00511
CALL JOB:SEARCH-R1
SET P0353 P0006
SFTON P0353
MOVL C00512 BC00512 V=250.0 PL=0
SFTOF
MOVL C00513 BC00513 V=500.0
'PRZEJAZD
MOVL C00514 BC00514 V=500.0
MOVJ C00515 BC00515 VJ=20.00
MOVJ C00516 BC00516 VJ=20.00
MOVL C00517 BC00517 V=500.0
MOVL C00518 BC00518 V=500.0
MOVL C00519 BC00519 V=500.0
'------------------------
'W29.11
'------------------------
MOVL C00520 BC00520 V=166.7 PL=0
REFP 3 C00521 BC00521
CALL JOB:SEARCH-R1
IMOV P0056 V=23.0 PL=0
SET P0354 P0006
SFTON P0354
REFP 3 C00522 BC00522
CALL JOB:SEARCH-R1
SET P0354 P0006
SFTON P0354
MOVL C00523 BC00523 V=250.0 PL=0
SFTOF
'PRZEJAZD
MOVL C00524 BC00524 V=500.0
'------------------------
'W29.14
'------------------------
MOVL C00525 BC00525 V=166.7 PL=0
REFP 3 C00526 BC00526
CALL JOB:SEARCH-R1
IMOV P0056 V=23.0 PL=0
SET P0355 P0006
SFTON P0355
REFP 3 C00527 BC00527
CALL JOB:SEARCH-R1
SET P0355 P0006
SFTON P0355
MOVL C00528 BC00528 V=250.0 PL=0
SFTOF
'PRZEJAZD
MOVL C00529 BC00529 V=500.0
'------------------------
'W63.17
'------------------------
MOVL C00530 BC00530 V=166.7 PL=0
REFP 3 C00531 BC00531
CALL JOB:SEARCH-R1
IMOV P0056 V=23.0 PL=0
SET P0356 P0006
SFTON P0356
REFP 3 C00532 BC00532
CALL JOB:SEARCH-R1
SET P0356 P0006
SFTON P0356
MOVL C00533 BC00533 V=250.0 PL=0
SFTOF
MOVL C00534 BC00534 V=500.0
MOVL C00535 BC00535 V=166.7 PL=0
REFP 3 C00536 BC00536
CALL JOB:SEARCH-R1
IMOV P0056 V=23.0 PL=0
SET P0357 P0006
SFTON P0357
REFP 3 C00537 BC00537
CALL JOB:SEARCH-R1
SET P0357 P0006
SFTON P0357
MOVL C00538 BC00538 V=250.0 PL=0
SFTOF
'PRZEJAZD
MOVL C00539 BC00539 V=500.0
MOVJ C00540 BC00540 VJ=30.00
MOVJ C00541 BC00541 VJ=30.00
MOVL C00542 BC00542 V=500.0
MOVL C00543 BC00543 V=500.0
'------------------------
'W62.20
'------------------------
MOVL C00544 BC00544 V=166.7 PL=0
REFP 3 C00545 BC00545
CALL JOB:SEARCH-R1
IMOV P0056 V=23.0 PL=0
SET P0358 P0006
SFTON P0358
REFP 3 C00546 BC00546
CALL JOB:SEARCH-R1
SET P0358 P0006
SFTON P0358
MOVL C00547 BC00547 V=250.0 PL=0
SFTOF
'PRZEJAZD
MOVL C00548 BC00548 V=500.0
'------------------------
'W63.23
'------------------------
MOVL C00549 BC00549 V=166.7 PL=0
REFP 3 C00550 BC00550
CALL JOB:SEARCH-R1
IMOV P0056 V=23.0 PL=0
SET P0359 P0006
SFTON P0359
REFP 3 C00551 BC00551
CALL JOB:SEARCH-R1
SET P0359 P0006
SFTON P0359
MOVL C00552 BC00552 V=250.0 PL=0
MOVL C00553 BC00553 V=500.0
'------------------------
'W29.29
'------------------------
MOVL C00554 BC00554 V=166.7 PL=0
REFP 3 C00555 BC00555
CALL JOB:SEARCH-R1
IMOV P0056 V=23.0 PL=0
SET P0360 P0006
SFTON P0360
REFP 3 C00556 BC00556
CALL JOB:SEARCH-R1
SET P0360 P0006
SFTON P0360
MOVL C00557 BC00557 V=250.0 PL=0
SFTOF
'PRZEJAZD
MOVL C00558 BC00558 V=500.0
MOVL C00559 BC00559 V=166.7 PL=0
REFP 3 C00560 BC00560
CALL JOB:SEARCH-R1
IMOV P0056 V=23.0 PL=0
SET P0361 P0006
SFTON P0361
REFP 3 C00561 BC00561
CALL JOB:SEARCH-R1
SET P0361 P0006
SFTON P0361
MOVL C00562 BC00562 V=250.0 PL=0
SFTOF
'------------------------
'W29.32
'------------------------
'PRZEJAZD
MOVL C00563 BC00563 V=500.0
MOVL C00564 BC00564 V=166.7 PL=0
REFP 3 C00565 BC00565
CALL JOB:SEARCH-R1
IMOV P0056 V=23.0 PL=0
SET P0362 P0006
SFTON P0362
REFP 3 C00566 BC00566
CALL JOB:SEARCH-R1
SET P0362 P0006
SFTON P0362
MOVL C00567 BC00567 V=250.0 PL=0
SFTOF
MOVL C00568 BC00568 V=500.0
MOVL C00569 BC00569 V=166.7 PL=0
REFP 3 C00570 BC00570
CALL JOB:SEARCH-R1
IMOV P0056 V=23.0 PL=0
SET P0363 P0006
SFTON P0363
REFP 3 C00571 BC00571
CALL JOB:SEARCH-R1
SET P0363 P0006
SFTON P0363
MOVL C00572 BC00572 V=250.0 PL=0
SFTOF
MOVL C00573 BC00573 V=500.0
MOVL C00574 BC00574 V=166.7 PL=0
REFP 3 C00575 BC00575
CALL JOB:SEARCH-R1
IMOV P0056 V=23.0 PL=0
SET P0364 P0006
SFTON P0364
REFP 3 C00576 BC00576
CALL JOB:SEARCH-R1
SET P0364 P0006
SFTON P0364
MOVL C00577 BC00577 V=250.0 PL=0
SFTOF
MOVJ C00578 BC00578 VJ=20.00
MOVJ C00579 BC00579 VJ=30.00
MOVJ C00580 BC00580 VJ=15.00
MOVJ C00581 BC00581 VJ=15.00
MOVL C00582 BC00582 V=166.7
MOVL C00583 BC00583 V=166.7 PL=0
REFP 3 C00584 BC00584
CALL JOB:SEARCH-R1
IMOV P0056 V=23.0 PL=0
SET P0365 P0006
SFTON P0365
REFP 3 C00585 BC00585
CALL JOB:SEARCH-R1
SET P0365 P0006
SFTON P0365
MOVL C00586 BC00586 V=250.0 PL=0
SFTOF
MOVL C00587 BC00587 V=166.7 PL=0
REFP 3 C00588 BC00588
CALL JOB:SEARCH-R1
IMOV P0056 V=23.0 PL=0
SET P0366 P0006
SFTON P0366
REFP 3 C00589 BC00589
CALL JOB:SEARCH-R1
SET P0366 P0006
SFTON P0366
MOVL C00590 BC00590 V=250.0 PL=0
SFTOF
MOVJ C00591 BC00591 VJ=20.00
MOVJ C00592 BC00592 VJ=30.00
MOVJ C00593 BC00593 VJ=30.00
'KONIEC SEARCH WEW STRONA
MOVJ C00594 BC00594 VJ=30.00
MOVJ C00595 BC00595 VJ=20.00
MOVJ C00596 BC00596 VJ=10.00
MOVJ C00597 BC00597 VJ=20.00
MOVJ C00598 BC00598 VJ=20.00
'------------------------
'W29.2
'------------------------
MOVL C00599 BC00599 V=500.0
'------------------------
'W63.5
MACRO1 MJ#(0) ARGF9
'------------------------
SFTOF
SFTON P0301
MOVL C00600 BC00600 V=166.7 PL=0
ARCON
MOVL C00601 BC00601 V=8.3
ARCOF
SFTOF
MOVL C00602 BC00602 V=500.0
MACRO1 MJ#(0) ARGF24
SFTON P0302
MOVL C00603 BC00603 V=166.7 PL=0
ARCON
MOVL C00604 BC00604 V=8.3
ARCOF
MOVL C00605 BC00605 V=166.7 PL=0
SFTOF
MOVL C00606 BC00606 V=500.0
SFTON P0303
MOVL C00607 BC00607 V=166.7 PL=0
ARCON
MOVL C00608 BC00608 V=8.3
ARCOF
SFTOF
MOVL C00609 BC00609 V=166.7 PL=0
MOVL C00610 BC00610 V=500.0
MOVJ C00611 BC00611 VJ=30.00
MOVJ C00612 BC00612 VJ=20.00
MOVJ C00613 BC00613 VJ=30.00
MOVJ C00614 BC00614 VJ=30.00
MOVL C00615 BC00615 V=500.0
'------------------------
'W29.14
'------------------------
SFTON P0304
MOVL C00616 BC00616 V=166.7 PL=0
ARCON
MOVL C00617 BC00617 V=8.3
ARCOF
MOVL C00618 BC00618 V=166.7 PL=0
SFTOF
'PRZEJAZD
MOVL C00619 BC00619 V=500.0
MOVL C00620 BC00620 V=500.0
'------------------------
'W63.17
'------------------------
SFTON P0305
MOVL C00621 BC00621 V=166.7 PL=0
ARCON
MOVL C00622 BC00622 V=8.3
ARCOF
MOVL C00623 BC00623 V=166.7 PL=0
SFTOF
MOVL C00624 BC00624 V=500.0
SFTON P0306
MOVL C00625 BC00625 V=166.7
ARCON
MOVL C00626 BC00626 V=8.3
ARCOF
MOVL C00627 BC00627 V=166.7 PL=0
SFTOF
'PRZEJAZD
MOVL C00628 BC00628 V=500.0
SFTON P0307
MOVL C00629 BC00629 V=166.7
ARCON
MOVL C00630 BC00630 V=8.3
ARCOF
MOVL C00631 BC00631 V=166.7 PL=0
SFTOF
MOVJ C00632 BC00632 VJ=20.00
MOVJ C00633 BC00633 VJ=20.00
MOVJ C00634 BC00634 VJ=30.00
MOVJ C00635 BC00635 VJ=30.00
MOVL C00636 BC00636 V=500.0
'------------------------
'W63.20
'------------------------
SFTON P0308
MOVL C00637 BC00637 V=166.7 PL=0
ARCON
MOVL C00638 BC00638 V=8.3
ARCOF
MOVL C00639 BC00639 V=166.7 PL=0
SFTOF
'PRZEJAZD
MOVL C00640 BC00640 V=500.0
'------------------------
'W63.23
'------------------------
SFTON P0309
MOVL C00641 BC00641 V=166.7 PL=0
ARCON
MOVL C00642 BC00642 V=8.3
ARCOF
MOVL C00643 BC00643 V=250.0 PL=0
SFTOF
MOVL C00644 BC00644 V=500.0
SFTON P0310
MOVL C00645 BC00645 V=166.7 PL=0
ARCON
MOVL C00646 BC00646 V=8.3
ARCOF
MOVL C00647 BC00647 V=250.0 PL=0
SFTOF
MOVL C00648 BC00648 V=500.0
SFTON P0311
MOVL C00649 BC00649 V=166.7 PL=0
ARCON
MOVL C00650 BC00650 V=8.3
ARCOF
MOVL C00651 BC00651 V=250.0 PL=0
SFTOF
MOVL C00652 BC00652 V=500.0
SFTON P0312
MOVL C00653 BC00653 V=166.7 PL=0
ARCON
MOVL C00654 BC00654 V=8.3
ARCOF
MOVL C00655 BC00655 V=250.0 PL=0
SFTOF
MOVL C00656 BC00656 V=500.0
SFTON P0313
MOVL C00657 BC00657 V=166.7 PL=0
ARCON
MOVL C00658 BC00658 V=8.3
ARCOF
MOVL C00659 BC00659 V=250.0 PL=0
SFTOF
MOVL C00660 BC00660 V=500.0
SFTON P0314
MOVL C00661 BC00661 V=166.7 PL=0
ARCON
MOVL C00662 BC00662 V=8.3
ARCOF
MOVL C00663 BC00663 V=250.0 PL=0
SFTOF
'PRZEJAZD
MOVL C00664 BC00664 V=333.3
'PRZEJAZD
'KONIEC SPAWANIA CZESCI WSPOLNEJ
MOVL C00665 BC00665 V=500.0
MOVL C00666 BC00666 V=500.0
MOVL C00667 BC00667 V=500.0
MOVL C00668 BC00668 V=333.3
MOVL C00669 BC00669 V=333.3
SFTON P0315
MOVL C00670 BC00670 V=166.7 PL=0
ARCON
MOVL C00671 BC00671 V=8.3
ARCOF
MOVL C00672 BC00672 V=250.0 PL=0
SFTOF
MOVL C00673 BC00673 V=333.3
SFTON P0316
MOVL C00674 BC00674 V=166.7 PL=0
ARCON
MOVL C00675 BC00675 V=8.3
ARCOF
MOVL C00676 BC00676 V=250.0 PL=0
SFTOF
MOVJ C00677 BC00677 VJ=10.00
MOVJ C00678 BC00678 VJ=10.00
MOVJ C00679 BC00679 VJ=30.00
MOVJ C00680 BC00680 VJ=20.00
MOVJ C00681 BC00681 VJ=50.00
MOVJ C00682 BC00682 VJ=20.00
MOVJ C00683 BC00683 VJ=10.00
MOVJ C00684 BC00684 VJ=20.00
MOVJ C00685 BC00685 VJ=20.00
'------------------------
'W28.2
'------------------------
MOVJ C00686 BC00686 VJ=10.00
MOVJ C00687 BC00687 VJ=10.00
MOVL C00688 BC00688 V=500.0
MOVL C00689 BC00689 V=500.0
'------------------------
'W62.5
'------------------------
SFTON P0351
MOVL C00690 BC00690 V=166.7 PL=0
ARCON
MOVL C00691 BC00691 V=8.3
ARCOF
MOVL C00692 BC00692 V=250.0 PL=0
SFTOF
'PRZEJAZD
MOVL C00693 BC00693 V=500.0
MOVL C00694 BC00694 V=500.0
MOVL C00695 BC00695 V=500.0
SFTON P0352
MOVL C00696 BC00696 V=166.7 PL=0
ARCON
MOVL C00697 BC00697 V=8.3
ARCOF
MOVL C00698 BC00698 V=250.0 PL=0
SFTOF
MOVL C00699 BC00699 V=500.0
'------------------------
'W29.8
'------------------------
SFTON P0353
MOVL C00700 BC00700 V=166.7 PL=0
ARCON
MOVL C00701 BC00701 V=8.3
ARCOF
MOVL C00702 BC00702 V=250.0 PL=0
SFTOF
MOVL C00703 BC00703 V=500.0
'PRZEJAZD
MOVL C00704 BC00704 V=500.0
MOVJ C00705 BC00705 VJ=20.00
MOVL C00706 BC00706 V=500.0
MOVL C00707 BC00707 V=500.0
MOVL C00708 BC00708 V=500.0
'------------------------
'W29.11
'------------------------
SFTON P0354
MOVL C00709 BC00709 V=166.7 PL=0
ARCON
MOVL C00710 BC00710 V=8.3
ARCOF
MOVL C00711 BC00711 V=250.0 PL=0
SFTOF
'PRZEJAZD
MOVL C00712 BC00712 V=500.0
'------------------------
'W29.14
'------------------------
SFTON P0355
MOVL C00713 BC00713 V=166.7 PL=0
ARCON
MOVL C00714 BC00714 V=8.3
ARCOF
MOVL C00715 BC00715 V=250.0 PL=0
SFTOF
'PRZEJAZD
MOVL C00716 BC00716 V=500.0
'------------------------
'W63.17
'------------------------
SFTON P0356
MOVL C00717 BC00717 V=166.7 PL=0
ARCON
MOVL C00718 BC00718 V=8.3
ARCOF
MOVL C00719 BC00719 V=250.0 PL=0
SFTOF
MOVL C00720 BC00720 V=500.0
SFTON P0357
MOVL C00721 BC00721 V=166.7 PL=0
ARCON
MOVL C00722 BC00722 V=8.3
ARCOF
MOVL C00723 BC00723 V=250.0 PL=0
SFTOF
'PRZEJAZD
MOVL C00724 BC00724 V=500.0
MOVJ C00725 BC00725 VJ=30.00
MOVJ C00726 BC00726 VJ=30.00
MOVJ C00727 BC00727 VJ=30.00
MOVL C00728 BC00728 V=500.0
MOVL C00729 BC00729 V=500.0
'------------------------
'W62.20
'------------------------
SFTON P0358
MOVL C00730 BC00730 V=166.7 PL=0
ARCON
MOVL C00731 BC00731 V=8.3
ARCOF
MOVL C00732 BC00732 V=250.0 PL=0
SFTOF
'PRZEJAZD
MOVL C00733 BC00733 V=500.0
'------------------------
'W63.23
'------------------------
SFTON P0359
MOVL C00734 BC00734 V=166.7 PL=0
ARCON
MOVL C00735 BC00735 V=8.3
ARCOF
MOVL C00736 BC00736 V=250.0 PL=0
MOVL C00737 BC00737 V=500.0
'------------------------
'W29.29
'------------------------
SFTON P0360
MOVL C00738 BC00738 V=166.7 PL=0
ARCON
MOVL C00739 BC00739 V=8.3
ARCOF
MOVL C00740 BC00740 V=250.0 PL=0
SFTOF
'PRZEJAZD
MOVL C00741 BC00741 V=500.0
SFTON P0361
MOVL C00742 BC00742 V=166.7 PL=0
ARCON
MOVL C00743 BC00743 V=8.3
ARCOF
MOVL C00744 BC00744 V=250.0 PL=0
SFTOF
MOVL C00745 BC00745 V=500.0
SFTON P0362
MOVL C00746 BC00746 V=166.7 PL=0
ARCON
MOVL C00747 BC00747 V=8.3
ARCOF
MOVL C00748 BC00748 V=250.0 PL=0
SFTOF
MOVL C00749 BC00749 V=500.0
SFTON P0363
MOVL C00750 BC00750 V=166.7 PL=0
ARCON
MOVL C00751 BC00751 V=8.3
ARCOF
MOVL C00752 BC00752 V=250.0 PL=0
SFTOF
MOVL C00753 BC00753 V=500.0
SFTON P0364
MOVL C00754 BC00754 V=166.7 PL=0
ARCON
MOVL C00755 BC00755 V=8.3
ARCOF
MOVL C00756 BC00756 V=250.0 PL=0
SFTOF
PAUSE
MOVJ C00757 BC00757 VJ=20.00
MOVJ C00758 BC00758 VJ=30.00
MOVJ C00759 BC00759 VJ=15.00
MOVJ C00760 BC00760 VJ=15.00
MOVL C00761 BC00761 V=166.7
MOVL C00762 BC00762 V=166.7
SFTON P0365
MOVL C00763 BC00763 V=83.3 PL=0
ARCON
MOVL C00764 BC00764 V=8.3
ARCOF
MOVL C00765 BC00765 V=250.0 PL=0
SFTOF
SFTON P0366
MOVL C00766 BC00766 V=166.7
MOVL C00767 BC00767 V=166.7 PL=0
ARCON
MOVL C00768 BC00768 V=8.3
ARCOF
MOVL C00769 BC00769 V=250.0 PL=0
SFTOF
MOVJ C00770 BC00770 VJ=20.00
MOVJ C00771 BC00771 VJ=30.00
MOVJ C00772 BC00772 VJ=30.00
CALL JOB:MOVE_OUT_OF_TUNNEL
END
